// TwinCAT 3 PLC project Calvin
// ProgramVersion: 3.1.4023.0
// libraries:
//   Tc2_ModbusRTU, * (Beckhoff Automation GmbH)
//   Tc2_SerialCom, * (Beckhoff Automation GmbH)
//   Tc2_Standard, * (Beckhoff Automation GmbH)
//   Tc2_System, * (Beckhoff Automation GmbH)
//   Tc2_Utilities, * (Beckhoff Automation GmbH)
//   Tc3_Interfaces, * (Beckhoff Automation GmbH)
//   Tc3_Module, * (Beckhoff Automation GmbH)
//   Tc2_OpcUa,3.3.2.0,Beckhoff Automation GmbH
// project tree:
//   Data types/ E_OffOn.TcDUT, E_Alarms.TcDUT, E_MachineState.TcDUT, E_MBState.TcDUT, E_Status.TcDUT
//   GVLs/ Global_Constants.TcGVL, Global_Alarms.TcGVL, Global_Points.TcGVL, Global_Variables.TcGVL, Global_Variables_Tags.TcGVL
//   / PlcTask.TcTTO
//   POUs/Functions/ F_AnalogIn.TcPOU, F_Current.TcPOU, F_Voltage.TcPOU, F_Temperature.TcPOU
//   POUs/Function_Blocks/ FB_Temp_Control.TcPOU
//   POUs/ MAIN.TcPOU, P_AlarmCheck.TcPOU, P_HeaterControl.TcPOU, P_State_Machine.TcPOU, P_VFD_Test.TcPOU
// real-time tasks:
//   TASK PlcTask: cycle T#10ms, priority 20, ADS port 350
// I/O:
//   DEVICE Device 1 (EtherCAT), AmsNetId 10.12.1.55.2.1
//     Term 1 (EK1200) [EK1200-5000 EtherCAT Power supply (2A E-Bus)]
//       Term 2 (EL3318) [EL3318 8Ch. Ana Input Thermocouple (TC)]
//       Term 3 (EL3318) [EL3318 8Ch. Ana Input Thermocouple (TC)]
//       Term 4 (EL3318) [EL3318 8Ch. Ana Input Thermocouple (TC)]
//       Term 5 (EL3314) [EL3314 4Ch. Ana. Input Thermocouple (TC)]
//       Term 6 (EL3058) [EL3058 8Ch. Ana. Input 4-20mA]
//       Term 7 (EL3058) [EL3058 8Ch. Ana. Input 4-20mA]
//       Term 8 (EL3058) [EL3058 8Ch. Ana. Input 4-20mA]
//       Term 9 (EL3058) [EL3058 8Ch. Ana. Input 4-20mA]
//       Term 10 (EL3058) [EL3058 8Ch. Ana. Input 4-20mA]
//       Term 11 (EL9410) [EL9410 E-Bus Power Supplier  (Diagnostics)]
//       Term 12 (EL4122) [EL4122 2Ch. Ana. Output  4-20mA, 16bit]
//       Term 13 (EL4122) [EL4122 2Ch. Ana. Output  4-20mA, 16bit]
//       Term 14 (EL4122) [EL4122 2Ch. Ana. Output  4-20mA, 16bit]
//       Term 15 (EL4122) [EL4122 2Ch. Ana. Output  4-20mA, 16bit]
//       Term 16 (EL4122) [EL4122 2Ch. Ana. Output  4-20mA, 16bit]
//       Term 17 (EL1889) [EL1889 16Ch. Dig. Input 24V, 3ms, negative]
//       Term 18 (EL1889) [EL1889 16Ch. Dig. Input 24V, 3ms, negative]
//       Term 19 (EL9410) [EL9410 E-Bus Power Supplier  (Diagnostics)]
//       Term 20 (EL2088) [EL2088 8Ch. Dig. Output 24V, 0.5A, switching to negative]
//       Term 21 (EL2088) [EL2088 8Ch. Dig. Output 24V, 0.5A, switching to negative]
//       Term 22 (EL2088) [EL2088 8Ch. Dig. Output 24V, 0.5A, switching to negative]
//       Term 23 (EL2088) [EL2088 8Ch. Dig. Output 24V, 0.5A, switching to negative]
//       Term 24 (EL2008) [EL2008 8Ch. Dig. Output 24V, 0.5A]
//       Term 25 (EL6021) [EL6021 Interface (RS422/485)]
//       Term 26 (EL6021) [EL6021 Interface (RS422/485)]
//       Term 27 (EL2008) [EL2008 8Ch. Dig. Output 24V, 0.5A]
//       Term 28 (EL9011) [EL9011 End Terminal]
//   DEVICE Device 2 (NOV-DP-RAM)
//     Box 29 (Retain Handler)
// variable links:
//   Calvin/Calvin Instance <-> Device 1 (EtherCAT)/Term 1 (EK1200)/Term 10 (EL3058)
//     PlcTask Inputs/Global_Variables.IT_3 <-> AI Standard Channel 1/Value
//     PlcTask Inputs/Global_Variables.VT_1 <-> AI Standard Channel 2/Value
//     PlcTask Inputs/Global_Variables.VT_2 <-> AI Standard Channel 3/Value
//     PlcTask Inputs/Global_Variables.VT_3 <-> AI Standard Channel 4/Value
//     PlcTask Inputs/Global_Variables.ZT_1302B <-> AI Standard Channel 5/Value
//   Calvin/Calvin Instance <-> Device 1 (EtherCAT)/Term 1 (EK1200)/Term 12 (EL4122)
//     PlcTask Outputs/Global_Variables.IP_1102A <-> Channel 1/Output
//     PlcTask Outputs/Global_Variables.IP_1102B <-> Channel 2/Output
//   Calvin/Calvin Instance <-> Device 1 (EtherCAT)/Term 1 (EK1200)/Term 13 (EL4122)
//     PlcTask Outputs/Global_Variables.HS_1102_Out <-> Channel 2/Output
//     PlcTask Outputs/Global_Variables.IP_1101 <-> Channel 1/Output
//   Calvin/Calvin Instance <-> Device 1 (EtherCAT)/Term 1 (EK1200)/Term 14 (EL4122)
//     PlcTask Outputs/Global_Variables.HT_2_CTRL <-> Channel 1/Output
//     PlcTask Outputs/Global_Variables.HT_3_CTRL <-> Channel 2/Output
//   Calvin/Calvin Instance <-> Device 1 (EtherCAT)/Term 1 (EK1200)/Term 15 (EL4122)
//     PlcTask Outputs/Global_Variables.HT_4_CTRL <-> Channel 1/Output
//     PlcTask Outputs/Global_Variables.HT_5_CTRL <-> Channel 2/Output
//   Calvin/Calvin Instance <-> Device 1 (EtherCAT)/Term 1 (EK1200)/Term 16 (EL4122)
//     PlcTask Outputs/Global_Variables.HT_6_CTRL <-> Channel 1/Output
//     PlcTask Outputs/Global_Variables.IP_1302B <-> Channel 2/Output
//   Calvin/Calvin Instance <-> Device 1 (EtherCAT)/Term 1 (EK1200)/Term 17 (EL1889)
//     PlcTask Inputs/Global_Variables.ZSH_1101A <-> Channel 4/Input
//     PlcTask Inputs/Global_Variables.ZSH_1103A <-> Channel 8/Input
//     PlcTask Inputs/Global_Variables.ZSH_1301A <-> Channel 14/Input
//     PlcTask Inputs/Global_Variables.ZSH_1302A <-> Channel 16/Input
//     PlcTask Inputs/Global_Variables.ZSH_1101B <-> Channel 6/Input
//     PlcTask Inputs/Global_Variables.ZSH_1103B <-> Channel 10/Input
//     PlcTask Inputs/Global_Variables.ZSH_1107 <-> Channel 2/Input
//     PlcTask Inputs/Global_Variables.ZSH_1300 <-> Channel 12/Input
//     PlcTask Inputs/Global_Variables.ZSL_1101A <-> Channel 3/Input
//     PlcTask Inputs/Global_Variables.ZSL_1103A <-> Channel 7/Input
//     PlcTask Inputs/Global_Variables.ZSL_1301A <-> Channel 13/Input
//     PlcTask Inputs/Global_Variables.ZSL_1302A <-> Channel 15/Input
//     PlcTask Inputs/Global_Variables.ZSL_1101B <-> Channel 5/Input
//     PlcTask Inputs/Global_Variables.ZSL_1103B <-> Channel 9/Input
//     PlcTask Inputs/Global_Variables.ZSL_1107 <-> Channel 1/Input
//     PlcTask Inputs/Global_Variables.ZSL_1300 <-> Channel 11/Input
//   Calvin/Calvin Instance <-> Device 1 (EtherCAT)/Term 1 (EK1200)/Term 18 (EL1889)
//     PlcTask Inputs/Global_Variables.LSH_1201 <-> Channel 6/Input
//     PlcTask Inputs/Global_Variables.LSH_1202 <-> Channel 8/Input
//     PlcTask Inputs/Global_Variables.LSH_1300A <-> Channel 12/Input
//     PlcTask Inputs/Global_Variables.LSL_1201 <-> Channel 5/Input
//     PlcTask Inputs/Global_Variables.LSL_1202 <-> Channel 7/Input
//     PlcTask Inputs/Global_Variables.LSL_1300A <-> Channel 11/Input
//     PlcTask Inputs/Global_Variables.ZSH_1104 <-> Channel 10/Input
//     PlcTask Inputs/Global_Variables.ZSH_1301B <-> Channel 4/Input
//     PlcTask Inputs/Global_Variables.ZSL_1104 <-> Channel 9/Input
//     PlcTask Inputs/Global_Variables.ZSL_1301B <-> Channel 3/Input
//   Calvin/Calvin Instance <-> Device 1 (EtherCAT)/Term 1 (EK1200)/Term 2 (EL3318)
//     PlcTask Inputs/Global_Variables.TI_1001 <-> TC Channel 6/Value
//     PlcTask Inputs/Global_Variables.TI_1101 <-> TC Channel 7/Value
//     PlcTask Inputs/Global_Variables.TI_1301 <-> TC Channel 8/Value
//     PlcTask Inputs/Global_Variables.TI_1001_Error <-> TC Channel 6/Status/Error
//     PlcTask Inputs/Global_Variables.TI_1101_Error <-> TC Channel 7/Status/Error
//     PlcTask Inputs/Global_Variables.TI_1301_Error <-> TC Channel 8/Status/Error
//     PlcTask Inputs/Global_Variables.TI_1100A <-> TC Channel 2/Value
//     PlcTask Inputs/Global_Variables.TI_1102A <-> TC Channel 1/Value
//     PlcTask Inputs/Global_Variables.TI_1100A_Error <-> TC Channel 2/Status/Error
//     PlcTask Inputs/Global_Variables.TI_1102A_Error <-> TC Channel 1/Status/Error
//     PlcTask Inputs/Global_Variables.TI_1100B <-> TC Channel 3/Value
//     PlcTask Inputs/Global_Variables.TI_1102B <-> TC Channel 5/Value
//     PlcTask Inputs/Global_Variables.TI_1100B_Error <-> TC Channel 3/Status/Error
//     PlcTask Inputs/Global_Variables.TI_1102B_Error <-> TC Channel 5/Status/Error
//     PlcTask Inputs/Global_Variables.TI_1100C <-> TC Channel 4/Value
//     PlcTask Inputs/Global_Variables.TI_1100C_Error <-> TC Channel 4/Status/Error
//   Calvin/Calvin Instance <-> Device 1 (EtherCAT)/Term 1 (EK1200)/Term 20 (EL2088)
//     PlcTask Outputs/Global_Variables.HS_1200 <-> Channel 3/Output
//     PlcTask Outputs/Global_Variables.HS_1201 <-> Channel 4/Output
//     PlcTask Outputs/Global_Variables.HS_1202 <-> Channel 7/Output
//     PlcTask Outputs/Global_Variables.HS_1301 <-> Channel 2/Output
//     PlcTask Outputs/Global_Variables.HS_1300A <-> Channel 8/Output
//     PlcTask Outputs/Global_Variables.HT_1_RELAY <-> Channel 5/Output
//     PlcTask Outputs/Global_Variables.HT_2_RELAY <-> Channel 6/Output
//     PlcTask Outputs/Global_Variables.YL_1001 <-> Channel 1/Output
//   Calvin/Calvin Instance <-> Device 1 (EtherCAT)/Term 1 (EK1200)/Term 21 (EL2088)
//     PlcTask Outputs/Global_Variables.HS_1101A <-> Channel 8/Output
//     PlcTask Outputs/Global_Variables.HS_1107 <-> Channel 7/Output
//     PlcTask Outputs/Global_Variables.HS_1203 <-> Channel 3/Output
//     PlcTask Outputs/Global_Variables.HS_1305 <-> Channel 4/Output
//     PlcTask Outputs/Global_Variables.HT_3_RELAY <-> Channel 1/Output
//     PlcTask Outputs/Global_Variables.HT_4_RELAY <-> Channel 2/Output
//     PlcTask Outputs/Global_Variables.HT_5_RELAY <-> Channel 5/Output
//     PlcTask Outputs/Global_Variables.HT_6_RELAY <-> Channel 6/Output
//   Calvin/Calvin Instance <-> Device 1 (EtherCAT)/Term 1 (EK1200)/Term 22 (EL2088)
//     PlcTask Outputs/Global_Variables.HS_1101B <-> Channel 1/Output
//     PlcTask Outputs/Global_Variables.HS_1103B <-> Channel 3/Output
//     PlcTask Outputs/Global_Variables.HS_1300B <-> Channel 4/Output
//     PlcTask Outputs/Global_Variables.HS_1301B <-> Channel 8/Output
//     PlcTask Outputs/Global_Variables.HS_1102_Enable <-> Channel 7/Output
//     PlcTask Outputs/Global_Variables.HS_1103A <-> Channel 2/Output
//     PlcTask Outputs/Global_Variables.HS_1301A <-> Channel 5/Output
//     PlcTask Outputs/Global_Variables.HS_1302A <-> Channel 6/Output
//   Calvin/Calvin Instance <-> Device 1 (EtherCAT)/Term 1 (EK1200)/Term 23 (EL2088)
//     PlcTask Outputs/Global_Variables.AI_1102A_Pump <-> Channel 1/Output
//     PlcTask Outputs/Global_Variables.AI_1102A_Solenoid <-> Channel 2/Output
//     PlcTask Outputs/Global_Variables.AI_1102B_Pump <-> Channel 3/Output
//     PlcTask Outputs/Global_Variables.AI_1102B_Solenoid <-> Channel 4/Output
//     PlcTask Outputs/Global_Variables.HS_1104 <-> Channel 5/Output
//     PlcTask Outputs/Global_Variables.SV_1201 <-> Channel 8/Output
//     PlcTask Outputs/Global_Variables.YL_1002 <-> Channel 6/Output
//   Calvin/Calvin Instance <-> Device 1 (EtherCAT)/Term 1 (EK1200)/Term 24 (EL2008)
//     PlcTask Outputs/Global_Variables.LED1_Buzzer <-> Channel 3/Output
//     PlcTask Outputs/Global_Variables.LED2_Buzzer <-> Channel 6/Output
//     PlcTask Outputs/Global_Variables.LED1_G <-> Channel 2/Output
//     PlcTask Outputs/Global_Variables.LED2_G <-> Channel 5/Output
//     PlcTask Outputs/Global_Variables.LED1_R <-> Channel 1/Output
//     PlcTask Outputs/Global_Variables.LED2_R <-> Channel 4/Output
//     PlcTask Outputs/Global_Variables.LED3_R <-> Channel 7/Output
//     PlcTask Outputs/Global_Variables.LED3_Y <-> Channel 8/Output
//   Calvin/Calvin Instance <-> Device 1 (EtherCAT)/Term 1 (EK1200)/Term 25 (EL6021)
//     PlcTask Inputs/P_State_Machine.MBV_Master.InData/D[{0..21}] <-> COM Inputs/Data In {0..21}  (22 links)
//     PlcTask Inputs/P_State_Machine.MBV_Master.InData/Status <-> COM Inputs/Status
//     PlcTask Outputs/P_State_Machine.MBV_Master.OutData/Ctrl <-> COM Outputs/Ctrl
//     PlcTask Outputs/P_State_Machine.MBV_Master.OutData/D[{0..21}] <-> COM Outputs/Data Out {0..21}  (22 links)
//   Calvin/Calvin Instance <-> Device 1 (EtherCAT)/Term 1 (EK1200)/Term 27 (EL2008)
//     PlcTask Outputs/Global_Variables.LED3_Buzzer <-> Channel 2/Output
//     PlcTask Outputs/Global_Variables.LED3_G <-> Channel 1/Output
//   Calvin/Calvin Instance <-> Device 1 (EtherCAT)/Term 1 (EK1200)/Term 3 (EL3318)
//     PlcTask Inputs/Global_Variables.TI_1 <-> TC Channel 4/Value
//     PlcTask Inputs/Global_Variables.TI_1302 <-> TC Channel 1/Value
//     PlcTask Inputs/Global_Variables.TI_1303 <-> TC Channel 2/Value
//     PlcTask Inputs/Global_Variables.TI_1304 <-> TC Channel 3/Value
//     PlcTask Inputs/Global_Variables.TI_2 <-> TC Channel 5/Value
//     PlcTask Inputs/Global_Variables.TI_3 <-> TC Channel 6/Value
//     PlcTask Inputs/Global_Variables.TI_4 <-> TC Channel 7/Value
//     PlcTask Inputs/Global_Variables.TI_5 <-> TC Channel 8/Value
//     PlcTask Inputs/Global_Variables.TI_1302_Error <-> TC Channel 1/Status/Error
//     PlcTask Inputs/Global_Variables.TI_1303_Error <-> TC Channel 2/Status/Error
//     PlcTask Inputs/Global_Variables.TI_1304_Error <-> TC Channel 3/Status/Error
//     PlcTask Inputs/Global_Variables.TI_1_Error <-> TC Channel 4/Status/Error
//     PlcTask Inputs/Global_Variables.TI_2_Error <-> TC Channel 5/Status/Error
//     PlcTask Inputs/Global_Variables.TI_3_Error <-> TC Channel 6/Status/Error
//     PlcTask Inputs/Global_Variables.TI_4_Error <-> TC Channel 7/Status/Error
//     PlcTask Inputs/Global_Variables.TI_5_Error <-> TC Channel 8/Status/Error
//   Calvin/Calvin Instance <-> Device 1 (EtherCAT)/Term 1 (EK1200)/Term 4 (EL3318)
//     PlcTask Inputs/Global_Variables.TI_{6..12} <-> TC Channel {1..7}/Value  (7 links)
//     PlcTask Inputs/Global_Variables.TI_{6..12}_Error <-> TC Channel {1..7}/Status/Error  (7 links)
//   Calvin/Calvin Instance <-> Device 1 (EtherCAT)/Term 1 (EK1200)/Term 5 (EL3314)
//     PlcTask Inputs/Global_Variables.TI_{1103..1106} <-> TC Inputs Channel {1..4}/Value  (4 links)
//     PlcTask Inputs/Global_Variables.TI_{1103..1106}_Error <-> TC Inputs Channel {1..4}/Status/Error  (4 links)
//   Calvin/Calvin Instance <-> Device 1 (EtherCAT)/Term 1 (EK1200)/Term 6 (EL3058)
//     PlcTask Inputs/Global_Variables.DPT_1100 <-> AI Standard Channel 1/Value
//     PlcTask Inputs/Global_Variables.DPT_1102A <-> AI Standard Channel 4/Value
//     PlcTask Inputs/Global_Variables.DPT_1102B <-> AI Standard Channel 5/Value
//     PlcTask Inputs/Global_Variables.PI_1001 <-> AI Standard Channel 6/Value
//     PlcTask Inputs/Global_Variables.PI_1100 <-> AI Standard Channel 2/Value
//     PlcTask Inputs/Global_Variables.PI_1101 <-> AI Standard Channel 3/Value
//     PlcTask Inputs/Global_Variables.PI_1200 <-> AI Standard Channel 7/Value
//     PlcTask Inputs/Global_Variables.PI_1300 <-> AI Standard Channel 8/Value
//   Calvin/Calvin Instance <-> Device 1 (EtherCAT)/Term 1 (EK1200)/Term 7 (EL3058)
//     PlcTask Inputs/Global_Variables.FIC_1102 <-> AI Standard Channel 1/Value
//     PlcTask Inputs/Global_Variables.FI_1001 <-> AI Standard Channel 2/Value
//     PlcTask Inputs/Global_Variables.FI_1300 <-> AI Standard Channel 5/Value
//     PlcTask Inputs/Global_Variables.FI_1301 <-> AI Standard Channel 4/Value
//     PlcTask Inputs/Global_Variables.FI_1200_1 <-> AI Standard Channel 3/Value
//     PlcTask Inputs/Global_Variables.ZT_1101 <-> AI Standard Channel 8/Value
//     PlcTask Inputs/Global_Variables.ZT_1102A <-> AI Standard Channel 6/Value
//     PlcTask Inputs/Global_Variables.ZT_1102B <-> AI Standard Channel 7/Value
//   Calvin/Calvin Instance <-> Device 1 (EtherCAT)/Term 1 (EK1200)/Term 8 (EL3058)
//     PlcTask Inputs/Global_Variables.AI_1102A <-> AI Standard Channel 3/Value
//     PlcTask Inputs/Global_Variables.AI_1102B <-> AI Standard Channel 4/Value
//     PlcTask Inputs/Global_Variables.AI_1301 <-> AI Standard Channel 5/Value
//     PlcTask Inputs/Global_Variables.LIC_1300 <-> AI Standard Channel 2/Value
//     PlcTask Inputs/Global_Variables.LI_1204 <-> AI Standard Channel 1/Value
//     PlcTask Inputs/Global_Variables.MI_1102A <-> AI Standard Channel 8/Value
//   Calvin/Calvin Instance <-> Device 1 (EtherCAT)/Term 1 (EK1200)/Term 9 (EL3058)
//     PlcTask Inputs/Global_Variables.FI_1200_2 <-> AI Standard Channel 1/Value
//     PlcTask Inputs/Global_Variables.FI_1200_3 <-> AI Standard Channel 2/Value
//     PlcTask Inputs/Global_Variables.FI_1201_1 <-> AI Standard Channel 4/Value
//     PlcTask Inputs/Global_Variables.FI_1201_2 <-> AI Standard Channel 5/Value
//     PlcTask Inputs/Global_Variables.FI_1201_3 <-> AI Standard Channel 6/Value
//     PlcTask Inputs/Global_Variables.IT_1 <-> AI Standard Channel 7/Value
//     PlcTask Inputs/Global_Variables.IT_2 <-> AI Standard Channel 8/Value
//     PlcTask Inputs/Global_Variables.MI_1102B <-> AI Standard Channel 3/Value
//   Calvin/Calvin Instance <-> Device 2 (NOV-DP-RAM)/Box 29 (Retain Handler)
//     PlcTask Retains/P_State_Machine.gpdiCycle_Count <-> Retains/P_State_Machine.gpdiCycle_Count_[851]

CONFIGURATION Calvin
    RESOURCE PLC ON TwinCAT3
        TASK PlcTask(INTERVAL := T#10ms, PRIORITY := 20);
        PROGRAM MAIN WITH PlcTask : MAIN;
    END_RESOURCE
END_CONFIGURATION

// ---- Data types/E_OffOn.TcDUT
// Calvin - E_OffOn
// Rev 1.00 - March 23, 2023

TYPE E_OffOn :
(
	eOFF 	:= 1,
	eON		:= 2
);
END_TYPE

// ---- Data types/E_Alarms.TcDUT
// Calvin - E_Alarms
// Rev 1.00 - May 25, 2023

TYPE E_Alarms :
(
	eNo_Alarms							:= 0,
	eWarmup_Alarm,					
	eEvacuation_Alarm,					
	eSteamBypass_Alarm,					
	eDesorption_Alarm,					
	eRepressurization_Alarm,					
	eAdsorption_Alarm,					
	eSystem_Alarm,					
	eTC_Alarm,					
	eT09_Alarm,					
	eT10_Alarm,					
	eT11_Alarm,					
	eT12_Alarm,					
	eT13_Alarm,					
	eT14_Alarm,					
	eT15_Alarm,					
	eT16_Alarm,					
	eT17_Alarm,					
	eT18_Alarm,					
	eT19_Alarm,					
	eT20_Alarm,					
	eTimeout_Alarm,							// 21		
	e22_Error,		
	eReactorBackflow_Error,			
	eEvacTargetPressure_Error,		
	eCondensateLS_Error,			
	eDesorpNominalPressure_Error,	
	eDesorpCO2Conc_Error,			
	eReactorCooling_Error,			
	eReactorHighPressure_Error,		
	eReactorLowPressure_Error,		
	eReactorHighTemp_Error,			
	eReactorLowTemp_Error,			
	eHighLevel_Error,				
	eLowLevel_Error,				
	eVacuumHighTemp_Error,			
	eCondenserNoFlow_Error,			
	eHeatTrace_Error,				
	eSteamLS_Error,					
	eHeatTraceTimeout_Error,		
	eDPT_311_Error,					
	eDPTError						
);                                  
END_TYPE

// ---- Data types/E_MachineState.TcDUT
// Calvin - E_MachineState
// Rev 1.00 - April 26, 2023

TYPE E_MachineState :
(
	eIdle						:= 0,
	eWarmup,
	eEvacuation,
	eSteamBypass,
	eDesorption,
	eRepressurization,
	eAdsorption,
	eReset,
	ePause,
	eSystemError
);
END_TYPE

// ---- Data types/E_MBState.TcDUT
// Calvin - E_MBState
// Rev 1.00 - April 6, 2023

TYPE E_MBState :
(
	eMBIdle			 			:= 0,
	eMBReadCoils,
	eMBReadInputStatus,
	eMBReadRegs,
	eMBReadInputRegs,
	eMBWriteSingleCoil,
	eMBWriteSingleReg,
	eMBWriteMultipleCoils,
	eMBWriteRegs
);
END_TYPE

// ---- Data types/E_Status.TcDUT
// Calvin - E_Status
// Rev 1.00 - April 27, 2023

TYPE E_Status :
(
	eStart_Warm_Up						:= 0,
	eWarmup_Running,							// 1
	eStart_Reactor_Reset,						// 2
	eSystem_Ready,								// 3
	eEvacuation_Running,						// 4
	eSteamBypass_Running,						// 5
	eRepressurization_Running,					// 6
	eDesorption_Running,						// 7
	eAdsorption_Running,						// 8
	e9,
	eStopping_Process,							// 10
	eStopping_Warmup,							// 11
	eStopping_Evacuation,						// 12
	eStopping_SteamBypass,						// 13
	eStopping_Repressurization,					// 14
	eStopping_Desorption,						// 15
	eStopping_Adsorption,						// 16
	e17,
	eCycle_Error,								// 18
	e19,
	e20,
	eTest_Running,								// 21
	eEvacuation_Process_Error,					// 22
	eSteamBypass_Process_Error,					// 23
	eRepressurization_Process_Error,			// 24
	eDesorption_Process_Error,					// 25
	eAdsorption_Process_Error,					// 26
	e27,
	e28,
	e29,
	eEvacuation_Complete,						// 30
	eSteamBypass_Complete,						// 31
	eRepressurization_Complete,					// 32
	eDesorption_Complete,						// 33
	eAdsorption_Complete						// 34
);
END_TYPE

// ---- GVLs/Global_Constants.TcGVL
// Calvin - Global_Constants
// Rev 1.00 - September 22, 2023

VAR_GLOBAL
	PID_CYCLE_TIME									: REAL 		:= 0.01;		// PID cycle time for heaters
	OUTPUT_MIN										: REAL		:= 200;			// Minimum output needed to energize solid state heater relay
	PERCENT_FACTOR									: REAL		:= 327.67;		// Factor to convert input to output percentage
	ALARM_COUNT										: INT		:= 100;			// Number of possible alarms
	PRESSURE_CUTOFF									: REAL		:= 0.8;
	DEFAULT_STEP_TIME								: REAL		:= 20000;		// 20 seconds default time
	SECONDS											: REAL		:= 1000;
	MINUTES											: REAL		:= 60000;
	RESET_TIME										: REAL		:= 2000;
	
	CONDENSER_LEVEL_REFILL							: REAL		:= 20;											// 09/21/23 PS
	CONDENSER_LEVEL_LOW_LIMIT						: REAL		:= 12;											// 09/21/23 PS
	CONDENSER_LEVEL_HIGH_LIMIT						: REAL		:= 60;											// 09/21/23 PS
	VACUUM_TANK_DRAIN_TIME							: REAL		:= 60;											// 09/22/23 PS
	
	MB_VFD_ENABLE_ADDR								: WORD		:= 8192;
	MB_VFD_FREQ_ADDR								: WORD		:= 8193;
	MB_VFD_BLOCK_ADDR								: WORD		:= 2315;
	MODBUS_TIMEOUT									: TIME 		:= T#1S;
	 
	BV_OPEN_MAX										: REAL		:= 100.0;                               	
	BV_OPEN_POS_THRESHOLD							: REAL		:= 10.0;			// Percent that valve must be within open position to trigger open status
	BV_CLOSED_POS_THRESHOLD							: REAL		:= 2;				// Percent that valve must be within closed position to trigger closed status
	                                					
END_VAR

// ---- GVLs/Global_Alarms.TcGVL
// Calvin - Global_Alarms
// Rev 1.00 - September 22, 2023

VAR_GLOBAL
	gbAlarmsLoaded									: BOOL;
	gbRunVFD										: BOOL;
	giActiveAlarm									: INT;
	gbAlarms										: ARRAY[0..100] OF BOOL;
	gsAlarms										: ARRAY[0..100] OF STRING;
	gsAlarmInfo										: ARRAY[0..100] OF STRING;
	gsTempAlarm										: STRING;

	gsTI_1101Error									: STRING	:= '-TI_1101 sensor error';						// 09/20/23 PS
	gsLowCondenserLevel								: STRING	:= '-Condenser level low';						// 09/07/23 PS
	gsTK1300HighLevel								: STRING	:= '-TK_1300 level high';
	
	gsBoilerPressureLow								: STRING	:= '-Boiler pressure low';
	gsDrainNotClear									: STRING	:= '-Drain not clear';
	gsValvesNotClosed								: STRING	:= '-Valves not closed';
	gsValvesNotOpen									: STRING	:= '-Valves not open';
	gsLRPCoolingFlowLow								: STRING	:= '-LRP cooling flow low';
	gsTargetPressureHigh							: STRING	:= '-Target pressure high';
	gsPI_1300OutOfRange								: STRING	:= '-PI_1300 out of range';
	gsPI_1100OutOfRange								: STRING	:= '-PI_1100 out of range';
	gsPI_1100PressureLow							: STRING	:= '-PI_1100 pressure low';
	gsPI_1101PressureLow							: STRING	:= '-PI_1101 pressure low';
	gsPI_1001PressureLow							: STRING	:= '-PI_1001 pressure low';
	gsVacuumLeak									: STRING	:= '-Vacuum leak';
	gsSteamFlowLow									: STRING	:= '-Steam flow low';
	gsSteamTempLow									: STRING	:= '-Steam temperature low';
	gsSteamTempError								: STRING	:= '-Steam temperature sensor error';
	gsLimitSwitchError								: STRING	:= '-Limit swtich error';
	gsValveOutOfRange								: STRING	:= '-Valve out of range';
	gsReactorPressureLow							: STRING	:= '-Reactor pressure low';
	gsThermocoupleError								: STRING	:= '-Thermocouple error';
	gsSorbentOverTemp								: STRING	:= '-Sorbent over temperature';
	gsTempOutOfRange								: STRING	:= '-Temperature out of range';
	gsNoAirFlow										: STRING	:= '-No air flow';
	gsCO2DifferentialError							: STRING	:= '-CO2 differential error';
	gsFanStillRunning								: STRING	:= '-Fan still runiing';
	gsFileSaveError									: STRING	:= 'File save error';
	
	ALARM_00										: STRING	:= '00/No Alarms';								// These must correspond to E_Alarms values
	ALARM_01										: STRING	:= '01/ Warmup Error - ';
	ALARM_02										: STRING	:= '02/ Evacuation Error - ';
	ALARM_03										: STRING	:= '03/ Steam Bypass Error - ';
	ALARM_04										: STRING	:= '04/ Desorption Error - ';
	ALARM_05										: STRING	:= '05/ Repressurization Error - ';
	ALARM_06										: STRING	:= '06/ Adsorption Error - ';
	ALARM_07										: STRING	:= '07/ System Error - ';
	ALARM_08										: STRING	:= '08/ Thermocouple Error';
	ALARM_09										: STRING	:= '09/Alarm';
	ALARM_10										: STRING	:= '10/Alarm';
	ALARM_11										: STRING	:= '11/Alarm';
	ALARM_12										: STRING	:= '12/Alarm';
	ALARM_13										: STRING	:= '13/Alarm';
	ALARM_14										: STRING	:= '14/Alarm';
	ALARM_15										: STRING	:= '15/Alarm';
	ALARM_16										: STRING	:= '16/Alarm';
	ALARM_17										: STRING	:= '17/Alarm';
	ALARM_18										: STRING	:= '18/Alarm';
	ALARM_19										: STRING	:= '19/Alarm';
	ALARM_20										: STRING	:= '20/Alarm';
	ALARM_21										: STRING	:= '21Timeout Error';
	ALARM_22										: STRING	:= '22Alarm';
	ALARM_23										: STRING	:= '23Alarm';
	ALARM_24										: STRING	:= '24Alarm';
	ALARM_25										: STRING	:= '25Alarm';
	ALARM_26										: STRING	:= '26Alarm';
	ALARM_27										: STRING	:= '27Alarm';
	ALARM_28										: STRING	:= '28Alarm';
	ALARM_29										: STRING	:= '29Alarm';
	ALARM_30										: STRING	:= '30Alarm';
	ALARM_31										: STRING	:= '31Alarm';
	ALARM_32										: STRING	:= '32Alarm';
	ALARM_33										: STRING	:= '33Alarm';
	ALARM_34										: STRING	:= '34Alarm';
	ALARM_35										: STRING	:= '35Alarm';
	ALARM_36										: STRING	:= '36Alarm';
	ALARM_37										: STRING	:= '37Alarm';
	ALARM_38										: STRING	:= '38Alarm';
	ALARM_39										: STRING	:= '39Alarm';
	ALARM_40										: STRING	:= '40Alarm';
	ALARM_41										: STRING	:= '41Alarm';
	ALARM_42										: STRING	:= '42Alarm';
	ALARM_43										: STRING	:= '43Alarm';
	ALARM_44										: STRING	:= '44Alarm';
	ALARM_45										: STRING	:= '45Alarm';
	ALARM_46										: STRING	:= '46Alarm';
	ALARM_47										: STRING	:= '47Alarm';
	ALARM_48										: STRING	:= '48Alarm';
	ALARM_49										: STRING	:= '49Alarm';
	ALARM_50										: STRING	:= '50Alarm';
END_VAR

// ---- GVLs/Global_Points.TcGVL
// Calvin - Global_Points
// Rev 1.00 - May 11, 2023

VAR_GLOBAL
	// Analog Input Sensor Ranges      			
	DPT_1102A_LOW									: REAL		:= 0.0;
	DPT_1102A_HIGH									: REAL		:= 10.0;
	DPT_1102A_MIN									: REAL		:= 0.01;
	DPT_1102A_OFFSET								: REAL		:= 0.0;
	FIC_1102_LOW									: REAL		:= 0.0;
	FIC_1102_HIGH									: REAL		:= 1500.0;
	FIC_1102_MIN									: REAL		:= 10.0;
	FIC_1102_OFFSET									: REAL		:= 0.0;
	AI_1102A_LOW									: REAL		:= 0.0;
	AI_1102A_HIGH									: REAL		:= 100.0;
	AI_1102A_MIN									: REAL		:= 0.01;
	AI_1102A_OFFSET									: REAL		:= 0.0;
	MI_1102A_LOW									: REAL		:= 0.0;
	MI_1102A_HIGH									: REAL		:= 100.0;
	MI_1102A_MIN									: REAL		:= 0.01;
	MI_1102A_OFFSET									: REAL		:= 0.0;
	ZT_1102A_LOW									: REAL		:= 0.0;
	ZT_1102A_HIGH									: REAL		:= 100.0;
	ZT_1102A_MIN									: REAL		:= 0.01;
	ZT_1102A_OFFSET									: REAL		:= 0.0;
	PI_1100_LOW										: REAL		:= 0.0;
	PI_1100_HIGH									: REAL		:= 100.0;
	PI_1100_MIN										: REAL		:= 0.01;
	PI_1100_OFFSET									: REAL		:= 0.0;
	DPT_1100_LOW									: REAL		:= -3.0;
	DPT_1100_HIGH									: REAL		:= 3.0;
	DPT_1100_MIN									: REAL		:= 0.01;
	DPT_1100_OFFSET									: REAL		:= 0.0;
	ZT_1102B_LOW									: REAL		:= 0.0;
	ZT_1102B_HIGH									: REAL		:= 100.0;
	ZT_1102B_MIN									: REAL		:= 0.01;
	ZT_1102B_OFFSET									: REAL		:= 0.0;
	AI_1102B_LOW									: REAL		:= 0.0;
	AI_1102B_HIGH									: REAL		:= 100.0;
	AI_1102B_MIN									: REAL		:= 0.01;
	AI_1102B_OFFSET									: REAL		:= 0.0;
	MI_1102B_LOW									: REAL		:= 0.0;
	MI_1102B_HIGH									: REAL		:= 100.0;
	MI_1102B_MIN									: REAL		:= 0.01;
	MI_1102B_OFFSET									: REAL		:= 0.0;
	DPT_1102B_LOW									: REAL		:= 0.0;
	DPT_1102B_HIGH									: REAL		:= 5.0;
	DPT_1102B_MIN									: REAL		:= 0.01;
	DPT_1102B_OFFSET								: REAL		:= 0.0;
	FI_1200_1_LOW									: REAL		:= 0.0;
	FI_1200_1_HIGH									: REAL		:= 1500.0;
	FI_1200_1_MIN									: REAL		:= 10.0;
	FI_1200_1_OFFSET								: REAL		:= 0.0;
	FI_1200_2_LOW									: REAL		:= 0.0;
	FI_1200_2_HIGH									: REAL		:= 1500.0;
	FI_1200_2_MIN									: REAL		:= 10.0;
	FI_1200_2_OFFSET								: REAL		:= 0.0;
	FI_1200_3_LOW									: REAL		:= 0.0;
	FI_1200_3_HIGH									: REAL		:= 1500.0;
	FI_1200_3_MIN									: REAL		:= 10.0;
	FI_1200_3_OFFSET								: REAL		:= 0.0;
	FI_1201_1_LOW									: REAL		:= 0.0;
	FI_1201_1_HIGH									: REAL		:= 1500.0;
	FI_1201_1_MIN									: REAL		:= 10.0;
	FI_1201_1_OFFSET								: REAL		:= 0.0;
	FI_1201_2_LOW									: REAL		:= 0.0;
	FI_1201_2_HIGH									: REAL		:= 1500.0;
	FI_1201_2_MIN									: REAL		:= 10.0;
	FI_1201_2_OFFSET								: REAL		:= 0.0;
	FI_1201_3_LOW									: REAL		:= 0.0;
	FI_1201_3_HIGH									: REAL		:= 1500.0;
	FI_1201_3_MIN									: REAL		:= 10.0;
	FI_1201_3_OFFSET								: REAL		:= 0.0;
	PI_1200_LOW										: REAL		:= 0.0;
	PI_1200_HIGH									: REAL		:= 100.0;
	PI_1200_MIN										: REAL		:= 0.01;
	PI_1200_OFFSET									: REAL		:= 0.0;
	PI_1001_LOW										: REAL		:= 0.0;
	PI_1001_HIGH									: REAL		:= 100.0;
	PI_1001_MIN										: REAL		:= 0.01;
	PI_1001_OFFSET									: REAL		:= 0.0;
	FI_1001_LOW										: REAL		:= 0.0;
	FI_1001_HIGH									: REAL		:= 100.0;
	FI_1001_MIN										: REAL		:= 0.01;
	FI_1001_OFFSET									: REAL		:= 0.0;
	ZT_1101_LOW										: REAL		:= 0.0;
	ZT_1101_HIGH									: REAL		:= 100.0;
	ZT_1101_MIN										: REAL		:= 0.01;
	ZT_1101_OFFSET									: REAL		:= 0.0;
	PI_1101_LOW										: REAL		:= 0.0;
	PI_1101_HIGH									: REAL		:= 100.0;
	PI_1101_MIN		 								: REAL		:= 0.01;
	PI_1101_OFFSET									: REAL		:= 0.0;
	LI_1204_LOW										: REAL		:= 0.0;
	LI_1204_HIGH									: REAL		:= 100.0;
	LI_1204_MIN										: REAL		:= 0.01;
	LI_1204_OFFSET									: REAL		:= 0.0;
	AI_1300_1_LOW									: REAL		:= 0.0;
	AI_1300_1_HIGH									: REAL		:= 100.0;
	AI_1300_1_MIN									: REAL		:= 0.01;
	AI_1300_1_OFFSET								: REAL		:= 0.0;
	AI_1300_2_LOW									: REAL		:= 0.0;
	AI_1300_2_HIGH									: REAL		:= 100.0;
	AI_1300_2_MIN									: REAL		:= 0.01;
	AI_1300_2_OFFSET								: REAL		:= 0.0;
	AI_1300_3_LOW									: REAL		:= 0.0;
	AI_1300_3_HIGH									: REAL		:= 100.0;
	AI_1300_3_MIN									: REAL		:= 0.01;
	AI_1300_3_OFFSET								: REAL		:= 0.0;
	PI_1300_LOW										: REAL		:= 0.0;
	PI_1300_HIGH									: REAL		:= 100.0;
	PI_1300_MIN										: REAL		:= 0.01;
	PI_1300_OFFSET									: REAL		:= 0.0;
	LIC_1300_LOW									: REAL		:= 0.0;
	LIC_1300_HIGH									: REAL		:= 100.0;
	LIC_1300_MIN									: REAL		:= 0.01;
	LIC_1300_OFFSET									: REAL		:= 0.0;
	FI_1300_LOW										: REAL		:= 0.0;
	FI_1300_HIGH									: REAL		:= 100.0;
	FI_1300_MIN										: REAL		:= 0.01;
	FI_1300_OFFSET									: REAL		:= 0.0;
	FI_1301_LOW										: REAL		:= 0.0;
	FI_1301_HIGH									: REAL		:= 100.0;
	FI_1301_MIN										: REAL		:= 0.01;
	FI_1301_OFFSET									: REAL		:= 0.0;
	AI_1301_LOW										: REAL		:= 0.0;
	AI_1301_HIGH									: REAL		:= 100.0;
	AI_1301_MIN										: REAL		:= 0.01;
	AI_1301_OFFSET									: REAL		:= 0.0;
	ZT_1302B_LOW									: REAL		:= 0.0;
	ZT_1302B_HIGH									: REAL		:= 0.0;
	ZT_1302B_MIN									: REAL		:= 0.0;
	ZT_1302B_OFFSET									: REAL		:= 0.0;
	
	MI_2001_LOW										: REAL		:= 0.0;
	MI_2001_HIGH									: REAL		:= 100.0;
	MI_2001_MIN										: REAL		:= 0.01;
	MI_2001_OFFSET									: REAL		:= 0.0;
	TI_2001_LOW										: REAL		:= 0.0;
	TI_2001_HIGH									: REAL		:= 100.0;
	TI_2001_MIN										: REAL		:= 0.01;
	TI_2001_OFFSET									: REAL		:= 0.0;
	SI_2001_LOW										: REAL		:= 0.0;
	SI_2001_HIGH									: REAL		:= 100.0;
	SI_2001_MIN										: REAL		:= 0.01;
	SI_2001_OFFSET									: REAL		:= 0.0;
	ZI_2001_LOW										: REAL		:= 0.0;
	ZI_2001_HIGH									: REAL		:= 100.0;
	ZI_2001_MIN										: REAL		:= 0.01;
	ZI_2001_OFFSET									: REAL		:= 0.0;
	PI_2001_LOW										: REAL		:= 0.0;
	PI_2001_HIGH									: REAL		:= 100.0;
	PI_2001_MIN										: REAL		:= 0.01;
	PI_2001_OFFSET									: REAL		:= 0.0;

	ZXI_2002_LOW									: REAL		:= 0.0;
	ZXI_2002_HIGH									: REAL		:= 100.0;
	ZXI_2002_MIN									: REAL		:= 0.01;
	ZXI_2002_OFFSET									: REAL		:= 0.0;
	ZYI_2002_LOW									: REAL		:= 0.0;
	ZYI_2002_HIGH									: REAL		:= 100.0;
	ZYI_2002_MIN									: REAL		:= 0.01;
	ZYI_2002_OFFSET									: REAL		:= 0.0;
                        				
END_VAR

// ---- GVLs/Global_Variables.TcGVL
// Calvin - Global_Variables
// Rev 1.00 - September 20, 2023

VAR_GLOBAL
	eState											: E_MachineState;

	grHS_1102Out									: REAL;
	grSteamValveSP									: REAL;
	gbVFDTest										: BOOL;
	gbReadMBVFD										: BOOL;
	gbReadMBWeather									: BOOL;
	gbReadMBInclinometer							: BOOL;
	gbHS_1102ValvesOpen								: BOOL;
	gbHS_1102ValvesClosed							: BOOL;
	gbVacuumHolding									: BOOL;

	datain					AT %I*					: REAL;
	dataout					AT %Q*					: BYTE;

	// Reactor
	DPT_1102A				AT %I*					: INT;			// Reactor Filter Differential Pressure (-7.46 to 7.46 mbar)
	FIC_1102				AT %I*					: INT;			// Reactor Air flow
	AI_1102A				AT %I*					: INT;			// Reactor Inlet C02 (ppm)
	AI_1102A_Pump			AT %Q*					: BOOL;			// Inlet CO2 pump
	AI_1102A_Solenoid		AT %Q*					: BOOL;			// Inlet CO2 solenoid
	MI_1102A				AT %I*					: INT;			// Reactor Inlet H20 (ppm)
	ZT_1102A				AT %I*					: INT;			// Reactor Inlet Isolation Valve Input
	PI_1100					AT %I*					: INT;			// Reactor Pressure
	TI_1102A				AT %I*					: INT;			// Reactor Inlet Temperature
	TI_1102A_Error			AT %I*					: BOOL;			// Reactor Inlet Temperature Error
	bTI_1102A_ErrActive								: BOOL;
	TI_1100A				AT %I*					: INT;			// Reactor Sorbent Temperature A
	TI_1100A_Error			AT %I*					: BOOL;			// Reactor Sorbent Temperature A Error
	bTI_1100A_ErrActive								: BOOL;
	TI_1100B				AT %I*					: INT;			// Reactor Sorbent Temperature B
	TI_1100B_Error			AT %I*					: BOOL;			// Reactor Sorbent Temperature B Error
	bTI_1100B_ErrActive								: BOOL;
	TI_1100C				AT %I*					: INT;			// Reactor Sorbent Temperature C
	TI_1100C_Error			AT %I*					: BOOL;			// Reactor Sorbent Temperature C Error
	bTI_1100C_ErrActive								: BOOL;
	DPT_1100				AT %I*					: INT;			// Reactor Differential Pressure
	ZT_1102B				AT %I*					: INT;			// Reactor Outlet Isolation Valve Input
	TI_1102B				AT %I*					: INT;			// Reactor Outlet Temperature
	TI_1102B_Error			AT %I*					: BOOL;			// Reactor Outlet Temperature Error
	bTI_1102B_ErrActive								: BOOL;
	AI_1102B				AT %I*					: INT;			// Reactor Outlet C02 (ppm)
	AI_1102B_Pump			AT %Q*					: BOOL;			// Outlet CO2 pump
	AI_1102B_Solenoid		AT %Q*					: BOOL;			// Outlet CO2 solenoid
	MI_1102B				AT %I*					: INT;			// Reactor Outlet H20 (ppm)
	DPT_1102B				AT %I*					: INT;			// Reactor Fan Static Pressure
	IP_1102A				AT %Q*					: INT;			// Reactor Inlet Isolation Butterfly Valve Output
	IP_1102B				AT %Q*					: INT;			// Reactor Outlet Isolation Butterfly Valve Output
	HS_1104					AT %Q*					: BOOL;			// Reactor valve
	ZSH_1104				AT %I*					: BOOL;			// Reactor valve open
	ZSL_1104				AT %I*					: BOOL;			// Reactor valve closed
	TI_1103					AT %I*					: INT;			// Reactor Wall Temperature 1
	TI_1103_Error			AT %I*					: BOOL;			// Reactor Wall Temperature 1 Error
	bTI_1103_ErrActive								: BOOL;
	TI_1104					AT %I*					: INT;			// Reactor Wall Temperature 1
	TI_1104_Error			AT %I*					: BOOL;			// Reactor Wall Temperature 1 Error
	bTI_1104_ErrActive								: BOOL;
	TI_1105					AT %I*					: INT;			// Reactor Wall Temperature 1
	TI_1105_Error			AT %I*					: BOOL;			// Reactor Wall Temperature 1 Error
	bTI_1105_ErrActive								: BOOL;
	TI_1106					AT %I*					: INT;			// Reactor Wall Temperature 1
	TI_1106_Error			AT %I*					: BOOL;			// Reactor Wall Temperature 1 Error
	bTI_1106_ErrActive								: BOOL;
	
	// Steam
	FI_1200_1				AT %I*					: INT;			// Boiler Feed Flow
	FI_1200_2				AT %I*					: INT;			// Boiler Feed Flow
	FI_1200_3				AT %I*					: INT;			// Boiler Feed Flow
	FI_1201_1				AT %I*					: INT;			// Boiler Feed Flow
	FI_1201_2				AT %I*					: INT;			// Boiler Feed Flow
	FI_1201_3				AT %I*					: INT;			// Boiler Feed Flow
	PI_1200					AT %I*					: INT;			// Boiler Feed Water Pressure
	PI_1001					AT %I*					: INT;			// Boiler Steam Pressure
	TI_1001					AT %I*					: INT;			// Boiler Steam Temperature
	TI_1001_Error			AT %I*					: BOOL;			// Boiler Steam Temperature Error
	bTI_1001_ErrActive								: BOOL;
	FI_1001					AT %I*					: INT;			// Steam Line Pressure
	ZT_1101					AT %I*					: INT;			// Steam Control Valve Input
	PI_1101					AT %I*					: INT;			// Steam Line Pressure
	TI_1101					AT %I*					: INT;			// Steam Line Temperature
	TI_1101_Error			AT %I*					: BOOL;			// Steam Line Temperature Error
	bTI_1101_ErrActive								: BOOL;
	ZSH_1107				AT %I*					: BOOL;			// Steam Bypass Valve High Limit Switch
	ZSL_1107				AT %I*					: BOOL;			// Steam Bypass Valve Low Limit Switch
	ZSH_1101A				AT %I*					: BOOL;			// Reactor Steam Isolation Valve A High Limit Switch
	ZSL_1101A				AT %I*					: BOOL;			// Reactor Steam Isolation Valve A Low Limit Switch
	ZSH_1101B				AT %I*					: BOOL;			// Reactor Steam Isolation Valve B High Limit Switch
	ZSL_1101B				AT %I*					: BOOL;			// Reactor Steam Isolation Valve B Low Limit Switch
	IP_1101					AT %Q*					: INT;			// Steam Control Valve Output
	YL_1001					AT %Q*					: BOOL;			// Boiler Power Contactor
	YL_1002					AT %Q*					: BOOL;			// Boiler Power Contactor
	HS_1107					AT %Q*					: BOOL;			// Steam Bypass Valve Output
	HS_1101A				AT %Q*					: BOOL;			// Reactor Steam Isolation Valve A
	HS_1101B				AT %Q*					: BOOL;			// Reactor Steam Isolation Valve B
	                                            	
	// Condensate
	HS_1201					AT %Q*					: BOOL;			// Reactor Drain Pump
	LSH_1201				AT %I*					: BOOL;			// Reactor Drain Level High
	LSL_1201				AT %I*					: BOOL;			// Reactor Drain Level Low
	HS_1103A				AT %Q*					: BOOL;			// Reactor To Vacuum Isolation Valve A
	ZSH_1103A				AT %I*					: BOOL;			// Reactor To Vacuum Isolation Valve A High Limit Switch
	ZSL_1103A				AT %I*					: BOOL;			// Reactor To Vacuum Isolation Valve A Low Limit Switch
	HS_1103B				AT %Q*					: BOOL;			// Reactor To Vacuum Isolation Valve B
	ZSH_1103B				AT %I*					: BOOL;			// Reactor To Vacuum Isolation Valve B High Limit Switch
	ZSL_1103B				AT %I*					: BOOL;			// Reactor To Vacuum Isolation Valve B Low Limit Switch
	HS_1203					AT %Q*					: BOOL;			// Condenser Heater Motor
	HS_1202					AT %Q*					: BOOL;			// Separator Drain Pump
	LSH_1202				AT %I*					: BOOL;			// Separator Drain Level High Switch
	LSL_1202				AT %I*					: BOOL;			// Separator Drain Level Low Switch
	LI_1204					AT %I*					: INT;			// Condensate Tank Level
	HS_1200					AT %Q*					: BOOL;			// Condensate/Boiler Feed Pump
	SV_1201					AT %Q*					: BOOL;			// Refill valve													// 09/19/23 PS
	ZSH_1202				AT %I*					: BOOL;			// Refill valve													// 09/19/23 PS
	ZSL_1202				AT %I*					: BOOL;			// Refill valve													// 09/19/23 PS
                                                	
	// Vacuum
	HS_1302A				AT %Q*					: BOOL;			// Vacuum Desorb Valve
	ZSH_1302A				AT %I*					: BOOL;			// Vacuum Desorb Valve High Limit Switch
	ZSL_1302A				AT %I*					: BOOL;			// Vacuum Desorb Valve Low Limit Switch
	IP_1302B				AT %Q*					: INT;			// Ambient Steam Desorption Valve
	ZT_1302B				AT %I*					: INT;			// Ambient Steam Desorption Valve feedback
	PI_1300					AT %I*					: INT;			// Vacuum System Pressure
	HS_1301A				AT %Q*					: BOOL;			// Eductor Valve
	ZSH_1301A				AT %I*					: BOOL;			// Eductor Valve High Limit Switch
	ZSL_1301A				AT %I*					: BOOL;			// Eductor Valve Low Limit Switch
	HS_1301B				AT %Q*					: BOOL;			// Vacuum Diverter Valve
	ZSH_1301B				AT %I*					: BOOL;			// Vacuum Diverter Valve High Limit Switch
	ZSL_1301B				AT %I*					: BOOL;			// Vacuum Diverter Valve Low Limit Switch
	TI_1303					AT %I*					: INT;			// Vacuum Temperature
	TI_1303_Error			AT %I*					: BOOL;			// Vacuum Temperature Error
	bTI_1303_ErrActive								: BOOL;
	HS_1301					AT %Q*					: BOOL;			// Vacuum Pump
	TI_1304					AT %I*					: INT;			// Vacuum Pump Outlet Temperature
	TI_1304_Error			AT %I*					: BOOL;			// Vacuum Pump Outlet Temperature Error
	bTI_1304_ErrActive								: BOOL;
	LIC_1300				AT %I*					: INT;			// Vacuum Pump Discharge Separation Level
	HS_1300B				AT %Q*					: BOOL;			// Automated Drain Valve
	ZSH_1300				AT %I*					: BOOL;			// Automated Drain Valve High Limit Switch
	ZSL_1300				AT %I*					: BOOL;			// Automated Drain Valve Low Limit Switch
	HS_1300A				AT %Q*					: BOOL;			// Vacuum Cooling Pump/Seal Water Circulation Pump
	LSH_1300A				AT %I*					: BOOL;			// Seal Water Circulation Pump Level High Switch
	LSL_1300A				AT %I*					: BOOL;			// Seal Water Circulation Pump Level Low Switch
	FI_1300					AT %I*					: INT;			// Flow Meter
	TI_1302					AT %I*					: INT;			// Vacuum Cooler Input Temperature
	TI_1302_Error			AT %I*					: BOOL;			// Vacuum Cooler Input Temperature Error
	bTI_1302_ErrActive								: BOOL;
	HS_1305					AT %Q*					: BOOL;			// Vacuum Cooler Motor
	TI_1301					AT %I*					: INT;			// Vacuum Cooler Output Temperature
	TI_1301_Error			AT %I*					: BOOL;			// Vacuum Cooler Output Temperature Error
	bTI_1301_ErrActive								: BOOL;
	FI_1301					AT %I*					: INT;			// CO2 Product Flow
	AI_1301					AT %I*					: INT;			// CO2 Product Purity

	// Heat Traces
	TI_1					AT %I*					: INT;			// Heat Trace 1 Temperature
	TI_1_Error				AT %I*					: BOOL;			// Heat Trace 1 Temperature Error
	bTI_1_ErrActive									: BOOL;
	TI_2					AT %I*					: INT;			// Heat Trace 2 Temperature
	TI_2_Error				AT %I*					: BOOL;			// Heat Trace 2 Temperature Error
	bTI_2_ErrActive									: BOOL;
	TI_3					AT %I*					: INT;			// Heat Trace 3 Temperature
	TI_3_Error				AT %I*					: BOOL;			// Heat Trace 3 Temperature Error
	bTI_3_ErrActive									: BOOL;
	TI_4					AT %I*					: INT;			// Heat Trace 4 Temperature
	TI_4_Error				AT %I*					: BOOL;			// Heat Trace 4 Temperature Error
	bTI_4_ErrActive									: BOOL;
	TI_5					AT %I*					: INT;			// Heat Trace 5 Temperature
	TI_5_Error				AT %I*					: BOOL;			// Heat Trace 5 Temperature Error
	bTI_5_ErrActive									: BOOL;
	TI_6					AT %I*					: INT;			// Heat Trace 6 Temperature
	TI_6_Error				AT %I*					: BOOL;			// Heat Trace 6 Temperature Error
	bTI_6_ErrActive									: BOOL;
	TI_7					AT %I*					: INT;			// Heat Trace 7 Temperature
	TI_7_Error				AT %I*					: BOOL;			// Heat Trace 7 Temperature Error
	bTI_7_ErrActive									: BOOL;
	TI_8					AT %I*					: INT;			// Heat Trace 8 Temperature
	TI_8_Error				AT %I*					: BOOL;			// Heat Trace 8 Temperature Error
	bTI_8_ErrActive									: BOOL;
	TI_9					AT %I*					: INT;			// Heat Trace 9 Temperature
	TI_9_Error				AT %I*					: BOOL;			// Heat Trace 9 Temperature Error
	bTI_09_ErrActive								: BOOL;
	TI_10					AT %I*					: INT;			// Heat Trace 10 Temperature
	TI_10_Error				AT %I*					: BOOL;			// Heat Trace 10 Temperature Error
	bTI_10_ErrActive								: BOOL;
	TI_11					AT %I*					: INT;			// Heat Trace 11 Temperature
	TI_11_Error				AT %I*					: BOOL;			// Heat Trace 11 Temperature Error
	bTI_11_ErrActive								: BOOL;
	TI_12					AT %I*					: INT;			// Heat Trace 12 Temperature
	TI_12_Error				AT %I*					: BOOL;			// Heat Trace 12 Temperature Error
	bTI_12_ErrActive	 							: BOOL;
	HT_1_RELAY				AT %Q*					: BOOL;
	HT_2_RELAY				AT %Q*					: BOOL;
	HT_3_RELAY				AT %Q*					: BOOL;
	HT_4_RELAY				AT %Q*					: BOOL;
	HT_5_RELAY				AT %Q*					: BOOL;
	HT_6_RELAY				AT %Q*					: BOOL;
	HT_1_CTRL				AT %Q*					: INT;
	HT_2_CTRL				AT %Q*					: INT;
	HT_3_CTRL				AT %Q*					: INT;
	HT_4_CTRL				AT %Q*					: INT;
	HT_5_CTRL				AT %Q*					: INT;
	HT_6_CTRL				AT %Q*					: INT;
	
	HS_1102_Enable			AT %Q*					: BOOL;
	HS_1102_Out				AT %Q*					: INT;					
	
	// Current & Voltage measuement
	IT_1					AT %I*					: INT;
	IT_2					AT %I*					: INT;
	IT_3					AT %I*					: INT;
	VT_1					AT %I*					: INT;
	VT_2					AT %I*					: INT;
	VT_3					AT %I*					: INT;
	
	// LED Outputs
	LED1_R					AT %Q*					: BOOL;
	LED1_G					AT %Q*					: BOOL;
	LED1_Buzzer				AT %Q*					: BOOL;
	LED2_R					AT %Q*					: BOOL;
	LED2_G					AT %Q*					: BOOL;
	LED2_Buzzer				AT %Q*					: BOOL;

	// Lightbar                                 	
	LED3_R					AT %Q*					: BOOL;
	LED3_Y					AT %Q*					: BOOL;
	LED3_G					AT %Q*					: BOOL;
	LED3_Buzzer				AT %Q*					: BOOL;
	
	// Weather Station
	MI_2001					AT %I*					: INT;
	TI_2001					AT %I*					: INT;
	SI_2001					AT %I*					: INT;
	ZI_2001					AT %I*					: INT;
	PI_2001					AT %I*					: INT;
	
	// Inclinometer
	ZXI_2002				AT %I*					: WORD;
	ZYI_2002				AT %I*					: WORD;
	                                            	
	LightBar_Green			AT %Q*					: BOOL;
	Lightbar_Yellow			AT %Q*					: BOOL;
	Lightbar_Red			AT %Q*					: BOOL;
	                                            	
END_VAR

// ---- GVLs/Global_Variables_Tags.TcGVL
// Calvin - Global_Variables_Tags
// Rev 1.00 - September 20, 2023

VAR_GLOBAL
	
	// {attribute 'OPC.UA.DA.Access' := '3'}			// 1=Read Only, 2=Write Only, 3=Read/Write (Default)
	tgs_Current_User								: STRING;																// 7/21/23 PS - Added current user for HMI control
	{attribute 'OPC.UA.DA' := '3'}  				
	tgi_Current_User_Level							: INT;																	// 7/21/23 PS - Added current user level for HMI control
	{attribute 'OPC.UA.DA' := '3'}  				
	tgb_Hmi_Locked									: BOOL;																	// 7/22/23 PS - Added current user level for HMI control
	{attribute 'OPC.UA.DA' := '3'}  				
	tgs_Hmi_Log_Date_Time							: STRING;																// 7/22/23 PS - Added current user level for HMI control

	{attribute 'OPC.UA.DA' := '3'}  				
	tgr_SP_Adsorption_Time							: REAL;
	{attribute 'OPC.UA.DA' := '3'}  				                
	tgr_SP_Adsorption_CO2_Differential				: REAL;
	{attribute 'OPC.UA.DA' := '3'}  				
	tgr_SP_Adsorption_CO2_Time						: REAL;
	{attribute 'OPC.UA.DA' := '3'}
	tgr_SP_Boiler_Temp								: REAL;
	{attribute 'OPC.UA.DA' := '3'}
	tgr_SP_Boiler_Pressure							: REAL;
	{attribute 'OPC.UA.DA' := '3'}  				                
	tgr_SP_Min_LRP_Cooling_Loop_Flow				: REAL;
	{attribute 'OPC.UA.DA' := '3'}  				                
	tgr_SP_Evacuation_Target_Pressure				: REAL;
	{attribute 'OPC.UA.DA' := '3'}  				                
	tgr_SP_Evacuation_Target_Pressure_Steam			: REAL;																	// 07/14/23 PS - Added set point
	{attribute 'OPC.UA.DA' := '3'}  				                
	tgr_SP_Max_Allowed_Pressure_Leakage				: REAL;
	{attribute 'OPC.UA.DA' := '3'}
	tgr_SP_Reactor_Repressurization_Pressure		: REAL;
	{attribute 'OPC.UA.DA' := '3'}  				
	tgr_SP_Adsorption_Temp							: REAL;
	{attribute 'OPC.UA.DA' := '3'}  				                
	tgr_SP_Adsorption_VFD_Output					: REAL;
	{attribute 'OPC.UA.DA' := '3'}  				                
	tgr_SP_Min_Bypass_Steam_Flow					: REAL;
	{attribute 'OPC.UA.DA' := '3'}  				                
	tgr_SP_Min_Bypass_Steam_Temp					: REAL;
	{attribute 'OPC.UA.DA' := '3'}  				
	tgr_SP_IP_1302B_Reactor_Low						: REAL;
	{attribute 'OPC.UA.DA' := '3'}  				      
	tgr_SP_IP_1302B_Reactor_High					: REAL;
	{attribute 'OPC.UA.DA' := '3'}  				      
	tgr_SP_IP_1302B_Valve_Low						: REAL;
	{attribute 'OPC.UA.DA' := '3'}  				      
	tgr_SP_IP_1302B_Valve_High						: REAL;
	{attribute 'OPC.UA.DA' := '3'}  				      
	tgr_SP_Steam_Valve_Percent_Open					: REAL;
	{attribute 'OPC.UA.DA' := '3'}  				      
	tgr_SP_Max_Allowed_Sorbent_Temp					: REAL;
	{attribute 'OPC.UA.DA' := '3'}                        
	tgr_SP_Steam_Repressurization_Pressure			: REAL;
	{attribute 'OPC.UA.DA' := '3'}                        
	tgr_SP_Steam_Purge_Time							: REAL;
	{attribute 'OPC.UA.DA' := '3'}                        
	tgr_SP_Steam_Purge_Cutoff_Temp					: REAL;
	{attribute 'OPC.UA.DA' := '3'}                        
	tgr_SP_Evap_Cooling_Cutoff_Temp					: REAL;
	{attribute 'OPC.UA.DA' := '3'}                        
	tgr_SP_Evap_Cooling_Target_Pressure				: REAL;
	{attribute 'OPC.UA.DA' := '3'}                        
	tgr_SP_Leak_Check_Time							: REAL;
	
	{attribute 'OPC.UA.DA' := '3'}  				                
	tgb_Warmup_Complete								: BOOL;
	{attribute 'OPC.UA.DA' := '3'}  				                
	tgb_HMI_Active									: BOOL;						// An HMI program is running and communicating
	{attribute 'OPC.UA.DA' := '2'}  				                
	tgb_Auto_Mode									: BOOL;						// Machine is in Auto Mode
	{attribute 'OPC.UA.DA' := '1'}  				                
	tgb_Watchdog									: BOOL;
	{attribute 'OPC.UA.DA' := '1'}  				                
	tgb_ADS_Active									: BOOL;						// ADS HMI program is running and communicating
	{attribute 'OPC.UA.DA' := '1'}  				
	tgb_Active_Alarm								: BOOL;
	{attribute 'OPC.UA.DA' := '3'}  				                
	tgb_Alarm_Reset									: BOOL;
	{attribute 'OPC.UA.DA' := '1'}  				
	tgb_Half_Sec_Pulse								: BOOL;
	{attribute 'OPC.UA.DA' := '3'}  				
	tgb_File_Save_Error								: BOOL;
	{attribute 'OPC.UA.DA' := '3'}  				                
	tgb_Test_Mode									: BOOL;						// Start or stop test
	{attribute 'OPC.UA.DA' := '1'}  				                
	tgb_Test_Running								: BOOL;						// Test is running
	{attribute 'OPC.UA.DA' := '1'}  				
	tgb_Stop_Cycle									: BOOL;
	{attribute 'OPC.UA.DA' := '1'}  				
	tgi_Current_Step								: INT;
	{attribute 'OPC.UA.DA' := '1'}  				
	tgi_Machine_State								: INT;
	{attribute 'OPC.UA.DA' := '1'}  				
	tgi_Alarm_State									: INT;						// Current Alarm State
	{attribute 'OPC.UA.DA' := '1'}  				
	tgi_Cycles_To_Run								: INT;
	{attribute 'OPC.UA.DA' := '1'}  				
	tgi_Cycle_Count									: INT;						// Number of TVSA cycles run since cycle restart
	{attribute 'OPC.UA.DA' := '1'}  				
	tgi_Status										: INT;
	{attribute 'OPC.UA.DA' := '1'}  				
	tgi_Total_Cycle_Count							: DINT;						// Total number of TVSA cycles run
	{attribute 'OPC.UA.DA' := '1'}  				
	tgr_Remaining_Time								: REAL;
	{attribute 'OPC.UA.DA' := '1'}  				
	tgs_Alarm										: STRING;
	{attribute 'OPC.UA.DA' := '1'}  				
	tgs_Active_Alarm								: STRING;
	{attribute 'OPC.UA.DA' := '1'}  				
	tgs_Status										: STRING;
	
	{attribute 'OPC.UA.DA' := '3'}  				
	tgb_Drains_On									: BOOL;
	{attribute 'OPC.UA.DA' := '3'}  				                
	tgb_Manual_Heater_Mode							: BOOL;						// Manual heater mode active
	{attribute 'OPC.UA.DA' := '1'}  				
	tgb_Adsorption_CO2								: BOOL;

	
	// Reactor
	{attribute 'OPC.UA.DA' := '1'}  				                
	tgr_DPT_1102A									: REAL;			
	{attribute 'OPC.UA.DA' := '1'}  				                
	tgr_FIC_1102									: REAL;			
	{attribute 'OPC.UA.DA' := '1'}  				                
	tgr_AI_1102A									: REAL;			
	{attribute 'OPC.UA.DA' := '3'}  				                
	tgb_AI_1102A_Pump								: BOOL;			
	{attribute 'OPC.UA.DA' := '1'}  				                
	tgb_AI_1102A_Pump_On							: BOOL;			
	{attribute 'OPC.UA.DA' := '3'}  				                
	tgb_AI_1102A_Solenoid							: BOOL;			
	{attribute 'OPC.UA.DA' := '1'}  				                
	tgb_AI_1102A_Solenoid_On						: BOOL;			
	{attribute 'OPC.UA.DA' := '1'}  				                
	tgr_MI_1102A									: REAL;			
	{attribute 'OPC.UA.DA' := '3'}  				                
	tgr_IP_1102A									: REAL;			
	{attribute 'OPC.UA.DA' := '3'}  				                
	tgr_IP_1102A_Output								: REAL;			
	{attribute 'OPC.UA.DA' := '1'}  				                
	tgr_ZT_1102A									: REAL;			
	{attribute 'OPC.UA.DA' := '1'}  				                
	tgr_PI_1100										: REAL;			
	{attribute 'OPC.UA.DA' := '1'}  				                
	tgr_DPT_1100									: REAL;			
	{attribute 'OPC.UA.DA' := '3'}  				                
	tgr_IP_1102B									: REAL;			
	{attribute 'OPC.UA.DA' := '3'}  				                
	tgr_IP_1102B_Output								: REAL;			
	{attribute 'OPC.UA.DA' := '1'}  				                
	tgr_ZT_1102B									: REAL;			
	{attribute 'OPC.UA.DA' := '1'}  				                
	tgr_AI_1102B									: REAL;			
	{attribute 'OPC.UA.DA' := '3'}  				                
	tgb_AI_1102B_Pump								: BOOL;			
	{attribute 'OPC.UA.DA' := '1'}  				                
	tgb_AI_1102B_Pump_On							: BOOL;			
	{attribute 'OPC.UA.DA' := '3'}  				                
	tgb_AI_1102B_Solenoid							: BOOL;			
	{attribute 'OPC.UA.DA' := '1'}  				                
	tgb_AI_1102B_Solenoid_On						: BOOL;			
	{attribute 'OPC.UA.DA' := '1'}  				                
	tgr_MI_1102B									: REAL;			
	{attribute 'OPC.UA.DA' := '1'}  				                
	tgr_DPT_1102B									: REAL;			
	{attribute 'OPC.UA.DA' := '1'}  				                
	tgr_TI_1102A									: REAL;			
	{attribute 'OPC.UA.DA' := '1'}  				                
	tgb_TI_1102A_Error								: BOOL;			
	{attribute 'OPC.UA.DA' := '1'}  				                
	tgr_TI_1100A									: REAL;			
	{attribute 'OPC.UA.DA' := '1'}  				                
	tgb_TI_1100A_Error								: BOOL;			
	{attribute 'OPC.UA.DA' := '1'}  				                
	tgr_TI_1100B									: REAL;			
	{attribute 'OPC.UA.DA' := '1'}  				                
	tgb_TI_1100B_Error								: BOOL;			
	{attribute 'OPC.UA.DA' := '1'}  				                
	tgr_TI_1100C									: REAL;			
	{attribute 'OPC.UA.DA' := '1'}  				                
	tgb_TI_1100C_Error								: BOOL;			
	{attribute 'OPC.UA.DA' := '1'}  				                
	tgr_TI_1102B									: REAL;			
	{attribute 'OPC.UA.DA' := '1'}  				                
	tgb_TI_1102B_Error								: BOOL;			

	{attribute 'OPC.UA.DA' := '3'}  				                
	tgr_HS_1102									: REAL;
	{attribute 'OPC.UA.DA' := '3'}  				                
	tgr_HS_1102_Output								: REAL;
	{attribute 'OPC.UA.DA' := '1'}  				                
	tgr_HS_1102_RPM									: REAL;			// Fan rpm
	{attribute 'OPC.UA.DA' := '1'}  				                
	tgr_HS_1102V									: REAL;			// VFD frequency
	{attribute 'OPC.UA.DA' := '1'}  				                
	tgb_HS_1102_Enabled								: BOOL;			// VFD enabled	
	{attribute 'OPC.UA.DA' := '1'}  				                
	tgb_HS_1102_Running								: BOOL;			// Fan running
	{attribute 'OPC.UA.DA' := '1'}  				                
	tgb_HS_1104										: BOOL;			
	{attribute 'OPC.UA.DA' := '1'}  				                
	tgb_HS_1104_On									: BOOL;			
	{attribute 'OPC.UA.DA' := '1'}  				                
	tgb_HS_1104_Open								: BOOL;			
	{attribute 'OPC.UA.DA' := '1'}  				                
	tgb_HS_1104_Closed								: BOOL;			
	
	{attribute 'OPC.UA.DA' := '1'}  				                
	tgb_IP_1102A_Open								: BOOL;			
	{attribute 'OPC.UA.DA' := '1'}  				                
	tgb_IP_1102A_Closed								: BOOL;			
	{attribute 'OPC.UA.DA' := '1'}  				                
	tgb_IP_1102B_Open								: BOOL;			
	{attribute 'OPC.UA.DA' := '1'}  				                
	tgb_IP_1102B_Closed								: BOOL;			
	{attribute 'OPC.UA.DA' := '3'}  				                
	tgb_YL_1001										: BOOL;			
	{attribute 'OPC.UA.DA' := '1'}  				                
	tgb_YL_1001_On									: BOOL;			

	{attribute 'OPC.UA.DA' := '1'}  				                
	tgr_FI_1200_1									: REAL;			
	{attribute 'OPC.UA.DA' := '1'}  				                
	tgr_FI_1200_2									: REAL;			
	{attribute 'OPC.UA.DA' := '1'}  				                
	tgr_FI_1200_3									: REAL;			
	{attribute 'OPC.UA.DA' := '1'}  				                
	tgr_FI_1201_1									: REAL;			
	{attribute 'OPC.UA.DA' := '1'}  				                
	tgr_FI_1201_2									: REAL;			
	{attribute 'OPC.UA.DA' := '1'}  				                
	tgr_FI_1201_3									: REAL;			
	{attribute 'OPC.UA.DA' := '1'}  				                
	tgr_PI_1200										: REAL;			
	{attribute 'OPC.UA.DA' := '1'}  				                
	tgr_PI_1001										: REAL;			
	{attribute 'OPC.UA.DA' := '1'}  				                
	tgr_TI_1001										: REAL;			
	{attribute 'OPC.UA.DA' := '1'}  				                
	tgb_TI_1001_Error								: BOOL;			
	{attribute 'OPC.UA.DA' := '1'}  				                
	tgr_FI_1001										: REAL;			
	{attribute 'OPC.UA.DA' := '3'}  				                
	tgr_IP_1101										: REAL;			
	{attribute 'OPC.UA.DA' := '3'}  				                
	tgr_IP_1101_Output								: REAL;			
	{attribute 'OPC.UA.DA' := '1'}  				                
	tgr_ZT_1101										: REAL;			
	{attribute 'OPC.UA.DA' := '1'}  				                
	tgr_PI_1101										: REAL;			
	{attribute 'OPC.UA.DA' := '1'}  				                
	tgr_TI_1101										: REAL;			
	{attribute 'OPC.UA.DA' := '1'}  				                
	tgb_TI_1101_Error								: BOOL;			
	{attribute 'OPC.UA.DA' := '3'}  				                
	tgb_HS_1107										: BOOL;			
	{attribute 'OPC.UA.DA' := '1'}  				                
	tgb_HS_1107_On									: BOOL;			
	{attribute 'OPC.UA.DA' := '1'}  				                
	tgb_HS_1107_Open								: BOOL;			
	{attribute 'OPC.UA.DA' := '1'}  				                
	tgb_HS_1107_Closed								: BOOL;			
	{attribute 'OPC.UA.DA' := '3'}  				                
	tgb_HS_1101A									: BOOL;			
	{attribute 'OPC.UA.DA' := '1'}  				                
	tgb_HS_1101A_On									: BOOL;			
	{attribute 'OPC.UA.DA' := '1'}  				                
	tgb_HS_1101A_Open								: BOOL;			
	{attribute 'OPC.UA.DA' := '1'}  				                
	tgb_HS_1101A_Closed								: BOOL;			
	{attribute 'OPC.UA.DA' := '3'}  				                
	tgb_HS_1101B									: BOOL;			
	{attribute 'OPC.UA.DA' := '1'}  				                
	tgb_HS_1101B_On									: BOOL;			
	{attribute 'OPC.UA.DA' := '1'}  				                
	tgb_HS_1101B_Open								: BOOL;			
	{attribute 'OPC.UA.DA' := '1'}  				                
	tgb_HS_1101B_Closed								: BOOL;			
	{attribute 'OPC.UA.DA' := '1'}  				                
	tgr_TI_1103										: REAL;			
	{attribute 'OPC.UA.DA' := '1'}  				                
	tgb_TI_1103_Error								: BOOL;			
	{attribute 'OPC.UA.DA' := '1'}  				                
	tgr_TI_1104										: REAL;			
	{attribute 'OPC.UA.DA' := '1'}  				                
	tgb_TI_1104_Error								: BOOL;			
	{attribute 'OPC.UA.DA' := '1'}  				                
	tgr_TI_1105										: REAL;			
	{attribute 'OPC.UA.DA' := '1'}  				                
	tgb_TI_1105_Error								: BOOL;			
	{attribute 'OPC.UA.DA' := '1'}  				                
	tgr_TI_1106										: REAL;			
	{attribute 'OPC.UA.DA' := '1'}  				                
	tgb_TI_1106_Error								: BOOL;			

	// Condensate
	{attribute 'OPC.UA.DA' := '3'}  				                
	tgb_HS_1201										: BOOL;			
	{attribute 'OPC.UA.DA' := '1'}  				                
	tgb_HS_1201_On									: BOOL;			
	{attribute 'OPC.UA.DA' := '1'}  				                
	tgb_HS_1201_LSH									: BOOL;			
	{attribute 'OPC.UA.DA' := '1'}  				                
	tgb_HS_1201_LSL									: BOOL;			
	{attribute 'OPC.UA.DA' := '3'}  				                
	tgb_HS_1103A									: BOOL;			
	{attribute 'OPC.UA.DA' := '1'}  				                
	tgb_HS_1103A_On									: BOOL;			
	{attribute 'OPC.UA.DA' := '1'}  				                
	tgb_HS_1103A_Open								: BOOL;			
	{attribute 'OPC.UA.DA' := '1'}  				                
	tgb_HS_1103A_Closed								: BOOL;			
	{attribute 'OPC.UA.DA' := '3'}  				                
	tgr_IP_1302B									: REAL;			
	{attribute 'OPC.UA.DA' := '3'}  				                
	tgr_IP_1302B_Output								: REAL;			
	{attribute 'OPC.UA.DA' := '1'}  				                
	tgr_ZT_1302B									: REAL;			
	{attribute 'OPC.UA.DA' := '3'}  				                
	tgb_HS_1103B									: BOOL;			
	{attribute 'OPC.UA.DA' := '1'}  				                
	tgb_HS_1103B_On									: BOOL;			
	{attribute 'OPC.UA.DA' := '1'}  				                
	tgb_HS_1103B_Open								: BOOL;			
	{attribute 'OPC.UA.DA' := '1'}  				                
	tgb_HS_1103B_Closed								: BOOL;			
	{attribute 'OPC.UA.DA' := '3'}  				                
	tgb_HS_1203										: BOOL;			
	{attribute 'OPC.UA.DA' := '3'}  				                
	tgb_HS_1203_On									: BOOL;			
	{attribute 'OPC.UA.DA' := '3'}  				                
	tgb_HS_1202										: BOOL;			
	{attribute 'OPC.UA.DA' := '1'}  				                
	tgb_HS_1202_On									: BOOL;			
	{attribute 'OPC.UA.DA' := '1'}  				                
	tgb_HS_1202_LSH									: BOOL;			
	{attribute 'OPC.UA.DA' := '1'}  				                
	tgb_HS_1202_LSL									: BOOL;			
	{attribute 'OPC.UA.DA' := '1'}  				                
	tgr_LI_1204										: REAL;			
	{attribute 'OPC.UA.DA' := '3'}  				                
	tgb_HS_1200										: BOOL;			
	{attribute 'OPC.UA.DA' := '1'}  				                
	tgb_HS_1200_On									: BOOL;			
	{attribute 'OPC.UA.DA' := '3'}  				                
	tgb_SV_1201										: BOOL;			
	{attribute 'OPC.UA.DA' := '1'}  				                
	tgb_SV_1201_On									: BOOL;			
	{attribute 'OPC.UA.DA' := '1'}  				                
	tgb_SV_1201_Open								: BOOL;			
	{attribute 'OPC.UA.DA' := '1'}  				                
	tgb_SV_1201_Closed								: BOOL;			
	
	// Vacuum
	{attribute 'OPC.UA.DA' := '1'}  				                
	tgr_AI_1300_1									: REAL;			
	{attribute 'OPC.UA.DA' := '1'}  				                
	tgr_AI_1300_2									: REAL;			
	{attribute 'OPC.UA.DA' := '1'}  				                
	tgr_AI_1300_3									: REAL;			
	{attribute 'OPC.UA.DA' := '3'}  				                
	tgb_HS_1302A									: BOOL;			
	{attribute 'OPC.UA.DA' := '1'}  				                
	tgb_HS_1302A_On									: BOOL;			
	{attribute 'OPC.UA.DA' := '1'}  				                
	tgb_HS_1302A_Open								: BOOL;			
	{attribute 'OPC.UA.DA' := '1'}  				                
	tgb_HS_1302A_Closed								: BOOL;			
	{attribute 'OPC.UA.DA' := '1'}  				                
	tgr_PI_1300										: REAL;			
	{attribute 'OPC.UA.DA' := '3'}  				                
	tgb_HS_1301A									: BOOL;			
	{attribute 'OPC.UA.DA' := '1'}  				                
	tgb_HS_1301A_On									: BOOL;			
	{attribute 'OPC.UA.DA' := '1'}  				                
	tgb_HS_1301A_Open								: BOOL;			
	{attribute 'OPC.UA.DA' := '1'}  				                
	tgb_HS_1301A_Closed								: BOOL;			
	{attribute 'OPC.UA.DA' := '3'}  				                
	tgb_HS_1301B									: BOOL;			
	{attribute 'OPC.UA.DA' := '1'}  				                
	tgb_HS_1301B_On									: BOOL;			
	{attribute 'OPC.UA.DA' := '1'}  				                
	tgb_HS_1301B_Open								: BOOL;			
	{attribute 'OPC.UA.DA' := '1'}  				                
	tgb_HS_1301B_Closed								: BOOL;			
	{attribute 'OPC.UA.DA' := '1'}  				                
	tgr_TI_1303										: REAL;			
	{attribute 'OPC.UA.DA' := '1'}  				                
	tgb_TI_1303_Error								: BOOL;
	{attribute 'OPC.UA.DA' := '3'}  				                
	tgb_HS_1301										: BOOL;			
	{attribute 'OPC.UA.DA' := '1'}  				                
	tgb_HS_1301_On									: BOOL;			
	{attribute 'OPC.UA.DA' := '1'}  				                
	tgr_TI_1304										: REAL;			
	{attribute 'OPC.UA.DA' := '1'}  				                
	tgb_TI_1304_Error								: BOOL;
	{attribute 'OPC.UA.DA' := '1'}  				                
	tgr_LIC_1300									: REAL;			
	{attribute 'OPC.UA.DA' := '3'}  				                
	tgb_HS_1300B									: BOOL;
	{attribute 'OPC.UA.DA' := '1'}  				                
	tgb_HS_1300B_On									: BOOL;
	{attribute 'OPC.UA.DA' := '1'}  				                
	tgb_HS_1300B_Open								: BOOL;			
	{attribute 'OPC.UA.DA' := '1'}  				                
	tgb_HS_1300B_Closed								: BOOL;			
	{attribute 'OPC.UA.DA' := '3'}  				                
	tgb_HS_1300A									: BOOL;			
	{attribute 'OPC.UA.DA' := '1'}  				                
	tgb_HS_1300A_On									: BOOL;			
	{attribute 'OPC.UA.DA' := '1'}  				                
	tgb_HS_1300A_LSH								: BOOL;			
	{attribute 'OPC.UA.DA' := '1'}  				                
	tgb_HS_1300A_LSL								: BOOL;			
	{attribute 'OPC.UA.DA' := '1'}  				                
	tgr_FI_1300										: REAL;			
	{attribute 'OPC.UA.DA' := '1'}  				                
	tgr_TI_1302										: REAL;			
	{attribute 'OPC.UA.DA' := '1'}  				                
	tgb_TI_1302_Error								: BOOL;			
	{attribute 'OPC.UA.DA' := '3'}  				                
	tgb_HS_1305										: BOOL;			
	{attribute 'OPC.UA.DA' := '1'}  				                
	tgb_HS_1305_On									: BOOL;			
	{attribute 'OPC.UA.DA' := '1'}  				                
	tgr_TI_1301										: REAL;			
	{attribute 'OPC.UA.DA' := '1'}  				                
	tgb_TI_1301_Error								: BOOL;			
	{attribute 'OPC.UA.DA' := '1'}  				                
	tgr_FI_1301										: REAL;			
	{attribute 'OPC.UA.DA' := '1'}  				                
	tgr_AI_1301										: REAL;			
				                                           
	// Heat Traces
	{attribute 'OPC.UA.DA' := '3'}  				                
	tgr_HT_P_Value									: REAL;						// Trace heater P factor
	{attribute 'OPC.UA.DA' := '3'}  				                
	tgr_HT_I_Value									: REAL;						// Trace heater I factor
	{attribute 'OPC.UA.DA' := '3'}  				                
	tgr_HT_I_Range									: REAL;						// Plus-minus range that Integral value is active in PID loop
	{attribute 'OPC.UA.DA' := '3'}  				                
	tgi_Manual_Heater_Output						: INT	:= 0;				// Manual heater output value
	{attribute 'OPC.UA.DA' := '1'}  				                
	tgr_TI_1										: REAL;			
	{attribute 'OPC.UA.DA' := '1'}  				                
	tgb_TI_1_Error									: BOOL;			
	{attribute 'OPC.UA.DA' := '3'}  				                
	tgb_HT_1_On										: BOOL;			
	{attribute 'OPC.UA.DA' := '3'}  				                
	tgr_HT_1_SP										: REAL;			
	{attribute 'OPC.UA.DA' := '1'}  				                
	tgr_HT_1_Ctrl									: REAL;			
	{attribute 'OPC.UA.DA' := '3'}  				                
	tgr_HT_1_Manual_Output							: REAL;			
	{attribute 'OPC.UA.DA' := '3'}  				                
	tgr_HT_1_Base_Output							: REAL;			
	{attribute 'OPC.UA.DA' := '1'}  				                
	tgr_TI_2										: REAL;			
	{attribute 'OPC.UA.DA' := '1'}  				                
	tgb_TI_2_Error									: BOOL;			
	{attribute 'OPC.UA.DA' := '3'}  				                
	tgb_HT_2_On										: BOOL;			
	{attribute 'OPC.UA.DA' := '3'}  				                
	tgr_HT_2_SP										: REAL;			
	{attribute 'OPC.UA.DA' := '1'}  				                
	tgr_HT_2_Ctrl									: REAL;			
	{attribute 'OPC.UA.DA' := '3'}  				                
	tgr_HT_2_Manual_Output							: REAL;			
	{attribute 'OPC.UA.DA' := '3'}  				                
	tgr_HT_2_Base_Output							: REAL;			
	{attribute 'OPC.UA.DA' := '1'}  				                
	tgr_TI_3										: REAL;			
	{attribute 'OPC.UA.DA' := '1'}  				                
	tgb_TI_3_Error									: BOOL;			
	{attribute 'OPC.UA.DA' := '3'}  				                
	tgb_HT_3_On										: BOOL;			
	{attribute 'OPC.UA.DA' := '3'}  				                
	tgr_HT_3_SP										: REAL;			
	{attribute 'OPC.UA.DA' := '1'}  				                
	tgr_HT_3_Ctrl									: REAL;			
	{attribute 'OPC.UA.DA' := '3'}  				                
	tgr_HT_3_Manual_Output							: REAL;			
	{attribute 'OPC.UA.DA' := '3'}  				                
	tgr_HT_3_Base_Output							: REAL;			
	{attribute 'OPC.UA.DA' := '1'}  				                
	tgr_TI_4										: REAL;			
	{attribute 'OPC.UA.DA' := '1'}  				                
	tgb_TI_4_Error									: BOOL;			
	{attribute 'OPC.UA.DA' := '3'}  				                
	tgb_HT_4_On										: BOOL;			
	{attribute 'OPC.UA.DA' := '3'}  				                
	tgr_HT_4_SP										: REAL;			
	{attribute 'OPC.UA.DA' := '1'}  				                
	tgr_HT_4_Ctrl									: REAL;			
	{attribute 'OPC.UA.DA' := '3'}  				                
	tgr_HT_4_Manual_Output							: REAL;			
	{attribute 'OPC.UA.DA' := '3'}  				                
	tgr_HT_4_Base_Output							: REAL;			
	{attribute 'OPC.UA.DA' := '1'}  				                
	tgr_TI_5										: REAL;			
	{attribute 'OPC.UA.DA' := '1'}  				                
	tgb_TI_5_Error									: BOOL;			
	{attribute 'OPC.UA.DA' := '3'}  				                
	tgb_HT_5_On										: BOOL;			
	{attribute 'OPC.UA.DA' := '3'}  				                
	tgr_HT_5_SP										: REAL;			
	{attribute 'OPC.UA.DA' := '1'}  				                
	tgr_HT_5_Ctrl									: REAL;			
	{attribute 'OPC.UA.DA' := '3'}  				                
	tgr_HT_5_Manual_Output							: REAL;			
	{attribute 'OPC.UA.DA' := '3'}  				                
	tgr_HT_5_Base_Output							: REAL;			
	{attribute 'OPC.UA.DA' := '1'}  				                
	tgr_TI_6										: REAL;			
	{attribute 'OPC.UA.DA' := '1'}  				                
	tgb_TI_6_Error									: BOOL;			
	{attribute 'OPC.UA.DA' := '3'}  				                
	tgb_HT_6_On										: BOOL;			
	{attribute 'OPC.UA.DA' := '3'}  				                
	tgr_HT_6_SP										: REAL;			
	{attribute 'OPC.UA.DA' := '1'}  				                
	tgr_HT_6_Ctrl									: REAL;			
	{attribute 'OPC.UA.DA' := '3'}  				                
	tgr_HT_6_Manual_Output							: REAL;			
	{attribute 'OPC.UA.DA' := '3'}  				                
	tgr_HT_6_Base_Output							: REAL;			
	{attribute 'OPC.UA.DA' := '1'}  				                
	tgr_TI_7										: REAL;			
	{attribute 'OPC.UA.DA' := '1'}  				                
	tgb_TI_7_Error									: BOOL;			
	{attribute 'OPC.UA.DA' := '1'}  				                
	tgr_TI_8										: REAL;			
	{attribute 'OPC.UA.DA' := '1'}  				                
	tgb_TI_8_Error									: BOOL;			
	{attribute 'OPC.UA.DA' := '1'}  				                
	tgr_TI_9										: REAL;			
	{attribute 'OPC.UA.DA' := '1'}  				                
	tgb_TI_9_Error									: BOOL;			
	{attribute 'OPC.UA.DA' := '1'}  				                
	tgr_TI_10										: REAL;			
	{attribute 'OPC.UA.DA' := '1'}  				                
	tgb_TI_10_Error									: BOOL;			
	{attribute 'OPC.UA.DA' := '1'}  				                
	tgr_TI_11										: REAL;			
	{attribute 'OPC.UA.DA' := '1'}  				                
	tgb_TI_11_Error									: BOOL;			
	{attribute 'OPC.UA.DA' := '1'}  				                
	tgr_TI_12										: REAL;			
	{attribute 'OPC.UA.DA' := '1'}  				                
	tgb_TI_12_Error									: BOOL;			
	
	// Current & Voltage
	{attribute 'OPC.UA.DA' := '1'}  				                
	tgr_IT_1										: REAL;			
	{attribute 'OPC.UA.DA' := '1'}  				                
	tgr_IT_2										: REAL;			
	{attribute 'OPC.UA.DA' := '1'}  				                
	tgr_IT_3										: REAL;			
	{attribute 'OPC.UA.DA' := '1'}  				                
	tgr_VT_1										: REAL;			
	{attribute 'OPC.UA.DA' := '1'}  				                
	tgr_VT_2										: REAL;			
	{attribute 'OPC.UA.DA' := '1'}  				                
	tgr_VT_3										: REAL;			
	
	
	// Weather Station
	{attribute 'OPC.UA.DA' := '1'}  				                
	tgr_MI_2001										: REAL;			
	{attribute 'OPC.UA.DA' := '1'}  				                
	tgr_TI_2001										: REAL;			
	{attribute 'OPC.UA.DA' := '1'}  				                
	tgr_SI_2001										: REAL;			
	{attribute 'OPC.UA.DA' := '1'}  				                
	tgr_ZI_2001										: REAL;			
	{attribute 'OPC.UA.DA' := '1'}  				                
	tgr_PI_2001										: REAL;			

	// Inclinometer  				                
	{attribute 'OPC.UA.DA' := '1'}
	tgr_ZXI_2002									: REAL;			
	{attribute 'OPC.UA.DA' := '1'}  				                
	tgr_ZYI_2002									: REAL;			
	
END_VAR

// ---- POUs/MAIN.TcPOU
PROGRAM MAIN

VAR
	rtrigHmiStartup									: R_TRIG;
	ftrigHmiShutdown								: F_TRIG;
	tonHalfSecPulse									: TON;
	tonWatchdog										: TON;
	bMBWeather										: BOOL;
	iVFDCount										: INT;
END_VAR

// Calvin - MAIN
// Rev 1.00 - August 5, 2023

P_State_Machine();
P_AlarmCheck();
P_HeaterControl();
P_VFD_Test();

rtrigHmiStartup(CLK:= tgb_ADS_Active);
IF rtrigHmiStartup.Q THEN
//	gbRunVFD										:= TRUE;
	tgr_HS_1102										:= 0;
END_IF
ftrigHmiShutdown(CLK:= tgb_ADS_Active);
IF ftrigHmiShutdown.Q THEN
//	gbRunVFD										:= FALSE;
	eState											:= eReset;
	P_State_Machine.A0_Reset();
END_IF

/// TIMER PULSE
IF tonHalfSecPulse.Q THEN
	tgb_Half_Sec_Pulse								:= NOT tgb_Half_Sec_Pulse;
	tgb_Watchdog									:= TRUE;
	tonHalfSecPulse(IN:= FALSE);
	iVFDCount										:= iVFDCount + 1;
	IF iVFDCount >= 4 THEN
		iVFDCount									:= 0;
		gbReadMBVFD									:= TRUE;
		IF bMBWeather THEN
			gbReadMBWeather							:= TRUE;
		ELSE
			gbReadMBInclinometer					:= TRUE;
		END_IF
		bMBWeather									:= NOT bMBWeather;
	END_IF
END_IF
tonHalfSecPulse(IN:= TRUE, PT:= T#500MS);

(*IF tonWatchdog.Q THEN
	tgb_ADS_Active									:= FALSE;
END_IF
tonWatchdog(IN:= tgb_Watchdog AND tgb_ADS_Active, PT:= T#4S);	*)

END_PROGRAM

// ---- POUs/P_State_Machine.TcPOU
PROGRAM P_State_Machine
VAR RETAIN
	gpdiCycle_Count									: DINT;
END_VAR
VAR
	strStatusLabel									: ARRAY[0..50] OF STRING;
	strError										: STRING;
	strProcessError									: STRING;
	bStatusListLoaded								: BOOL;	
	
	rtrigWarmup										: R_TRIG;
	rtrigEvacuation									: R_TRIG;
	rtrigSteamBypass								: R_TRIG;
	rtrigDesorption									: R_TRIG;
	rtrigRepressurization							: R_TRIG;
	rtrigAdsorption									: R_TRIG;
	rtrigStatusReady								: R_TRIG;

	iStep											: INT;
	i1Step											: INT;
	i2Step											: INT;
	i3Step											: INT;
	i4Step											: INT;
	i5Step											: INT;
	i6Step											: INT;
	
	bVacuumHolding									: BOOL;
	bWarmUpDone										: BOOL;
	bRunEvacuation									: BOOL;
	bEvacuationDone									: BOOL;
	bSteamBypassDone								: BOOL;
	bDesorptionDone							        : BOOL;
	bRepressurizationDone							: BOOL;
	bAdsorptionDone									: BOOL;
	bRunning										: BOOL;
	bInRange1										: BOOL;
	bInRange2										: BOOL;
	bInRange3										: BOOL;
	bTempAGood										: BOOL;
	bTempBGood										: BOOL;
	bTempCGood										: BOOL;
	bOverTemp										: BOOL;
	bStop											: BOOL;
	bTimer1											: BOOL;
	bTimer2											: BOOL;
	rTime1											: REAL;
	rTime2											: REAL;
	rSP1											: REAL;
	rSP2											: REAL;
	tonTimer1										: TON;
	tonTimer2										: TON;
	tonReset										: TON;
	tonPause										: TON;

	bRunValveModulation								: BOOL;
	bValveInRange									: BOOL;
	bFanError										: BOOL;
	bClearDrains									: BOOL;
	bCondenserLow									: BOOL;				// 09/07/23 PS
	bCondenserFull									: BOOL;				// 09/19/23 PS
	bCondenserRefill								: BOOL;				// 09/21/23 PS
	rOut											: REAL;
	rPI_1100_Save									: REAL;
	
	bDrainLSHClear									: BOOL;
	bDrainLSLClear									: BOOL;
	b1200DrainOROff									: BOOL;				// AF_Drains 4/7/23
	b1201DrainOn									: BOOL;				// AF_Drains 4/7/23
	b1202DrainOn									: BOOL;				// AF_Drains 4/7/23
	b1300DrainOn									: BOOL;				// 09/21/23 PS
	bDrainOn										: BOOL;				// AF_Drains 4/7/23
	b1201DrainOROff									: BOOL;				// 09/20/23 PS
	b1202DrainOROff									: BOOL;				// 09/20/23 PS
	b1202DrainOROn									: BOOL;				// 09/20/23 PS
	rtrigDrainsOff									: R_TRIG;			// 09/20/23 PS
	
	// A_DPT_Fan_Test
	tonFanTest										: TON;
	rtrigFanTest									: R_TRIG;
	ftrigFanTest									: F_TRIG;	
	tFanTestTime									: TIME	:= T#60S;
	rHS_1102										: REAL	:= 0.0;
	rFanIncrement									: REAL	:= 10.0;
	rFanMaximum										: REAL	:= 100.0;
	iFanTestStep									: INT	:= 0;
	bFanTimer										: BOOL;

	// A_Modbus_VFD
	MBV_Master 										: ModbusRtuMasterV2_KL6x22B;	
	MBV_Errors										: MODBUS_ERRORS;
	tonMBVReset										: TON;
	bMBVBusy										: BOOL;
	bMBVError										: BOOL;
	bMBVReadStatus									: BOOL;
	bMBVStatusCheck									: BOOL;
	iMBVFunction									: INT;
	iMBVHzRetry										: INT;
	uiMBVRead										: UINT;	
	wMBVAddress										: WORD;
	wMBVQuantity									: WORD;
	wMBVOnOff										: WORD;
	wMBVStatus										: WORD 	:= 3;
	wMBVReadData 									: ARRAY[0..21] OF WORD;
	wMBVWriteData 									: ARRAY[0..21] OF WORD;
	// A_Modbus_Points
	MBP_Master 										: ModbusRtuMasterV2_KL6x22B;	
	MBP_Errors										: MODBUS_ERRORS;
	tonMBPReset										: TON;
	bMBPWeather										: BOOL;
	bMBPBusy										: BOOL;
	bMBPError										: BOOL;
	iMBPFunction									: INT;
	uiMBPRead										: UINT;	
	wMBPAddress										: WORD;
	wMBPQuantity									: WORD;
	wMBPReadData 									: ARRAY[0..21] OF WORD;
	wMBPWriteData 									: ARRAY[0..21] OF WORD;

END_VAR

// Calvin - P_State_Machine
// Rev 1.00 - September 21, 2023

IF NOT bStatusListLoaded THEN
	A_Status_List();
END_IF

A_Temperatures();																											// Run these actions continuously
A_Inputs_Outputs();
A_Interlocks();
A_Modbus_VFD();
//A_Modbus_Points();
A_DPT_Fan_Test();
A_WaterHandling();

rtrigWarmup(CLK:= tgi_Machine_State = eWarmup);																				// Set trigger (one shot) on initial entry of each state
rtrigEvacuation(CLK:= tgi_Machine_State = eEvacuation);
rtrigSteamBypass(CLK:= tgi_Machine_State = eSteamBypass);
rtrigDesorption(CLK:= tgi_Machine_State = eDesorption);
rtrigRepressurization(CLK:= tgi_Machine_State = eRepressurization);
rtrigAdsorption(CLK:= tgi_Machine_State = eAdsorption);

IF rtrigWarmup.Q THEN																										// Warm up triggered
	bWarmUpDone										:= FALSE;																// Clear Done flag
	i1Step											:= 1;
	eState											:= eWarmup;																// Set state
ELSIF rtrigEvacuation.Q THEN
	bEvacuationDone									:= FALSE;
	i2Step											:= 1;
	eState											:= eEvacuation;
ELSIF rtrigSteamBypass.Q THEN
	bSteamBypassDone								:= FALSE;
	i3Step											:= 1;
	eState											:= eSteamBypass;
ELSIF rtrigDesorption.Q THEN
	bDesorptionDone									:= FALSE;
	i4Step											:= 1;
	eState											:= eDesorption;
ELSIF rtrigRepressurization.Q THEN
	bRepressurizationDone							:= FALSE;
	i5Step											:= 1;
	eState											:= eRepressurization;
ELSIF rtrigAdsorption.Q THEN																								// Adsorption triggered
	bAdsorptionDone									:= FALSE;																// Clear Done flag
	bFanError										:= FALSE;
	i6Step											:= 1;																	// Start Adsorption Case statement
	eState											:= eAdsorption;															// Set state
END_IF

bDrainOn 											:= eState >= eWarmup AND eState <= eAdsorption;							// Turn on drain function

CASE eState OF
	
	eIdle:
		tgi_Machine_State							:= eIdle;																// Indicate state to HMI
		tgb_Auto_Mode								:= FALSE;																// Clear flags
		tgb_Stop_Cycle								:= FALSE;
		i1Step										:= 0;
		i2Step										:= 0;
		i3Step										:= 0;
		i4Step										:= 0;
		i5Step										:= 0;
		i6Step										:= 0;
		tgi_Current_Step							:= 0;
		IF bRunEvacuation THEN
			tgi_Machine_State						:= eEvacuation;
		ELSE
			tgi_Status								:= SEL(tgb_Test_Running, SEL(NOT tgb_Warmup_Complete, eSystem_Ready, eStart_Warm_Up), eTest_Running);
		END_IF
		
	eWarmup:
		tgi_Status									:= SEL(bStop, eWarmup_Running, eStopping_Warmup);
		IF tgb_Stop_Cycle THEN																							
			bStop									:= TRUE;
		ELSIF bWarmUpDone THEN																								// Process complete
			bStop									:= FALSE;
			IF tgb_Warmup_Complete THEN
				eState								:= eIdle;																// Return to manual state
			ELSE
				eState								:= ePause;																// User stopped - allow status string to be displayed momentarily
			END_IF	
		END_IF
		
	eEvacuation:
		tgi_Status									:= SEL(bStop, eEvacuation_Running, SEL(tgb_Auto_Mode, eStopping_Evacuation, eStopping_Process));
		IF tgb_Stop_Cycle THEN
			bStop									:= TRUE;			
		ELSIF bEvacuationDone THEN
			IF tgb_Auto_Mode THEN
				tgi_Machine_State					:= eSteamBypass;
			ELSE
				IF bStop THEN
					bStop							:= FALSE;
					eState							:= eIdle;
				ELSE
					tgi_Status						:= eEvacuation_Complete;
					bRunEvacuation					:= FALSE;
					eState							:= ePause;
				END_IF
			END_IF
		END_IF
		
	eSteamBypass:
		tgi_Status									:= SEL(bStop, eSteamBypass_Running, SEL(tgb_Auto_Mode, eStopping_SteamBypass, eStopping_Process));
		IF tgb_Stop_Cycle THEN
			bStop									:= TRUE;
		ELSIF bSteamBypassDone THEN
			IF tgb_Auto_Mode THEN
				tgi_Machine_State					:= eDesorption;
			ELSE
				IF bStop THEN
					bStop							:= FALSE;
					eState							:= eIdle;
				ELSE
					tgi_Status						:= eSteamBypass_Complete;
					eState							:= ePause;
				END_IF
			END_IF
		END_IF
		
	eDesorption:
		tgi_Status									:= SEL(bStop, eDesorption_Running, SEL(tgb_Auto_Mode, eStopping_Desorption, eStopping_Process));
		IF tgb_Stop_Cycle THEN
			bStop									:= TRUE;
		ELSIF bDesorptionDone THEN
			IF tgb_Auto_Mode THEN
				tgi_Machine_State					:= eRepressurization;
			ELSE
				IF bStop THEN
					bStop							:= FALSE;
					eState							:= eIdle;
				ELSE
					tgi_Status						:= eDesorption_Complete;
					eState							:= ePause;
				END_IF
			END_IF
		END_IF
		
	eRepressurization:
		tgi_Status									:= SEL(bStop, eRepressurization_Running, SEL(tgb_Auto_Mode, eStopping_Repressurization, eStopping_Process));
		IF tgb_Stop_Cycle THEN
			bStop									:= TRUE;
		ELSIF bRepressurizationDone THEN
			IF tgb_Auto_Mode THEN
				tgi_Machine_State					:= eAdsorption;
			ELSE
				IF bStop THEN
					bStop							:= FALSE;
					eState							:= eIdle;
				ELSE
					tgi_Status						:= eRepressurization_Complete;
					eState							:= ePause;
				END_IF
			END_IF
		END_IF
		
	eAdsorption:
		tgi_Status									:= SEL(bStop, eAdsorption_Running, SEL(tgb_Auto_Mode, eStopping_Adsorption, eStopping_Process));
		IF tgb_Stop_Cycle THEN
			bStop									:= TRUE;
		ELSIF bAdsorptionDone THEN
			IF tgb_Auto_Mode THEN
				tgi_Cycle_Count						:= tgi_Cycle_Count + 1;
				gpdiCycle_Count						:= gpdiCycle_Count + 1;
				IF tgi_Cycle_Count >= tgi_Cycles_To_Run THEN
					eState							:= eIdle;
				ELSE
					tgi_Machine_State				:= eEvacuation;
				END_IF
			ELSE
				IF bFanError THEN
					tgi_Machine_State				:= eEvacuation;
				ELSIF bStop THEN
					bStop							:= FALSE;
					eState							:= eIdle;
				ELSIF bRunEvacuation THEN
					eState							:= eIdle;
				ELSE
					tgi_Status						:= eAdsorption_Complete;
					eState							:= ePause;
				END_IF
			END_IF
		END_IF
		
	eReset:
		IF tonReset.Q THEN
			A0_Reset();
			eState									:= eIdle;
		END_IF

	ePause:
		tgi_Machine_State							:= ePause;
		IF tonPause.Q THEN
			eState									:= eIdle;
		END_IF
		
	eSystemError:
		;
		
END_CASE

CASE tgi_Alarm_State OF
	
	1: ;																					// Level 1 alarm 
	
	2: ;																					// Level 2 alarm
	
	3: 	tgb_Stop_Cycle								:= TRUE;								// Level 3 alarm - stop cycle but no reset
		tgi_Alarm_State								:= 5;
	
	4:	tgb_Warmup_Complete							:= FALSE;								// Level 4 alarm - reset everything
		A0_Reset();
		tgi_Alarm_State								:= 5;
		eState										:= eSystemError;

	5:	 ;
	
END_CASE

rtrigStatusReady(CLK:= tgb_Warmup_Complete);
IF rtrigStatusReady.Q THEN
	tgi_Status										:= eSystem_Ready;
END_IF

A1_WarmUp();																										// Run action for this state
A2_Evacuation();
A3_SteamBypass();
A4_Desorption();
A5_Repressurization();
A6_Adsorption();

tonTimer1(IN:= bTimer1, PT:= REAL_TO_TIME(rTime1));
tonTimer2(IN:= bTimer2, PT:= REAL_TO_TIME(rTime2));

IF i1Step + i2Step + i3Step + i4Step + i5Step + i6Step > 0 THEN
	IF bTimer1 THEN
		tgr_Remaining_Time							:= rTime1 - TIME_TO_REAL(tonTimer1.ET);
	ELSIF bTimer2 THEN
		tgr_Remaining_Time							:= rTime2 - TIME_TO_REAL(tonTimer2.ET);
	ELSE
		tgr_Remaining_Time							:= 0;
	END_IF
END_IF

tgs_Status											:= strStatusLabel[tgi_Status];
bRunning											:= eState > eIdle AND eState < eReset;									// 09/19/23 PS
gbVFDTest											:= SEL(bRunning, gbVFDTest, FALSE);										// 09/19/23 PS
tgb_Drains_On										:= SEL(tgb_Auto_Mode, tgb_Drains_On, FALSE);							// 09/19/23 PS

tonReset(IN:= eState = eReset, PT:= REAL_TO_TIME(RESET_TIME));
tonPause(IN:= eState = ePause, PT:= REAL_TO_TIME(RESET_TIME));

ACTION A_ClearProcess:
// Calvin - A_ClearProcess
// Rev 1.00 - September 22, 2023

IF giActiveAlarm > 0 THEN
	gsAlarmInfo[giActiveAlarm]				:= CONCAT(INT_TO_STRING(iStep), strError);
	gbAlarmsLoaded							:= FALSE;
END_IF
bTimer1								 		:= FALSE;
bTimer2								 		:= FALSE;
tgb_Stop_Cycle								:= FALSE;
tgb_Auto_Mode								:= FALSE;
END_ACTION

ACTION A_DPT_Fan_Test:
// Calvin - A_DPT_Fan_Test
// Rev 1.00 - July 14, 2023

rtrigFanTest(CLK:= tgb_Test_Mode);
ftrigFanTest(CLK:= tgb_Test_Mode);

IF rtrigFanTest.Q THEN
	iFanTestStep									:= 1;
END_IF
IF ftrigFanTest.Q THEN
	iFanTestStep									:= 4;
END_IF

CASE iFanTestStep OF
	
	0:	tgb_Test_Running							:= FALSE;

	1:	tgr_IP_1102A								:= 100;
		tgr_IP_1102B								:= 100;
		tgb_Test_Running							:= TRUE;
		rFanIncrement								:= 10;
		tgr_HS_1102									:= 0;
		iFanTestStep								:= 2;
	
	2:	IF tgb_IP_1102A_Open AND tgb_IP_1102B_Open THEN
			bFanTimer								:= TRUE;
			tgr_HS_1102								:= rFanIncrement;
			iFanTestStep							:= 3;
		END_IF
		
	3:	;
	
	4:	bFanTimer									:= FALSE;
		tgr_HS_1102									:= 0;
		IF tgr_HS_1102_RPM = 0 THEN
			tgr_IP_1102A							:= 0;
			tgr_IP_1102B							:= 0;
			iFanTestStep							:= 0;
		END_IF

END_CASE;

IF tonFanTest.Q THEN
	tgr_HS_1102										:= tgr_HS_1102 + rFanIncrement;
	IF tgr_HS_1102 > rFanMaximum THEN
		rFanIncrement								:= 0 - rFanIncrement;
		tgr_HS_1102									:= rFanMaximum + rFanIncrement;
	ELSIF tgr_HS_1102 <= 0 THEN
		tgb_Test_Mode								:= FALSE;
	END_IF
	
	tonFanTest(IN:= FALSE);
END_IF

tonFanTest(IN:= bFanTimer, PT:= tFanTestTime);
END_ACTION

ACTION A_Inputs_Outputs:
// Calvin - A_Inputs_Outputs
// Rev 1.00 - September 20, 2023

//// DIGITAL IN
tgb_HS_1104_Open									:= ZSH_1104;			
tgb_HS_1104_Closed									:= ZSL_1104;				
tgb_HS_1107_Open									:= ZSH_1107;			
tgb_HS_1107_Closed									:= ZSL_1107;				
tgb_HS_1101A_Open									:= ZSH_1101A;				
tgb_HS_1101A_Closed									:= ZSL_1101A;				
tgb_HS_1101B_Open									:= ZSH_1101B;				
tgb_HS_1101B_Closed									:= ZSL_1101B;			
tgb_HS_1201_LSH										:= LSH_1201;					
tgb_HS_1201_LSL										:= LSL_1201;					
tgb_HS_1103A_Open									:= ZSH_1103A;				
tgb_HS_1103A_Closed									:= ZSL_1103A;				
tgb_HS_1103B_Open									:= ZSH_1103B;				
tgb_HS_1103B_Closed									:= ZSL_1103B;				
tgb_HS_1202_LSH										:= LSH_1202;			
tgb_HS_1202_LSL										:= LSL_1202;				
tgb_HS_1302A_Open									:= ZSH_1302A;			
tgb_HS_1302A_Closed									:= ZSL_1302A;			
tgb_HS_1301A_Open									:= ZSH_1301A;				
tgb_HS_1301A_Closed									:= ZSL_1301A;				
tgb_HS_1301B_Open									:= ZSH_1301B;				
tgb_HS_1301B_Closed									:= ZSL_1301B;				
tgb_HS_1300B_Open									:= ZSH_1300;					
tgb_HS_1300B_Closed									:= ZSL_1300;					
tgb_HS_1300A_LSH									:= LSH_1300A;			
tgb_HS_1300A_LSL									:= LSL_1300A;				
tgb_SV_1201_Open									:= ZSH_1202;				
tgb_SV_1201_Closed									:= ZSL_1202;				

//// ANALOG IN
tgr_DPT_1102A										:= F_AnalogIn(DPT_1102A, DPT_1102A_LOW, DPT_1102A_HIGH, DPT_1102A_MIN, DPT_1102A_OFFSET);
tgr_FIC_1102										:= F_AnalogIn(FIC_1102, FIC_1102_LOW, FIC_1102_HIGH, FIC_1102_MIN, FIC_1102_OFFSET);
tgr_AI_1102A										:= F_AnalogIn(AI_1102A, AI_1102A_LOW, AI_1102A_HIGH, AI_1102A_MIN, AI_1102A_OFFSET);
tgr_MI_1102A										:= F_AnalogIn(MI_1102A, MI_1102A_LOW, MI_1102A_HIGH, MI_1102A_MIN, MI_1102A_OFFSET);
tgr_ZT_1102A										:= F_AnalogIn(ZT_1102A, ZT_1102A_LOW, ZT_1102A_HIGH, ZT_1102A_MIN, ZT_1102A_OFFSET);
tgr_PI_1100											:= F_AnalogIn(PI_1100, PI_1100_LOW, PI_1100_HIGH, PI_1100_MIN, PI_1100_OFFSET);
tgr_DPT_1100										:= F_AnalogIn(DPT_1100, DPT_1100_LOW, DPT_1100_HIGH, DPT_1100_MIN, DPT_1100_OFFSET);
tgr_ZT_1102B										:= F_AnalogIn(ZT_1102B, ZT_1102B_LOW, ZT_1102B_HIGH, ZT_1102B_MIN, ZT_1102B_OFFSET);
tgr_AI_1102B										:= F_AnalogIn(AI_1102B, AI_1102B_LOW, AI_1102B_HIGH, AI_1102B_MIN, AI_1102B_OFFSET);
tgr_MI_1102B										:= F_AnalogIn(MI_1102B, MI_1102B_LOW, MI_1102B_HIGH, MI_1102B_MIN, MI_1102B_OFFSET);
tgr_DPT_1102B										:= F_AnalogIn(DPT_1102B, DPT_1102B_LOW, DPT_1102B_HIGH, DPT_1102B_MIN, DPT_1102B_OFFSET);
tgr_FI_1200_1										:= F_AnalogIn(FI_1200_1, FI_1200_1_LOW, FI_1200_1_HIGH, FI_1200_1_MIN, FI_1200_1_OFFSET);
tgr_FI_1200_2										:= F_AnalogIn(FI_1200_2, FI_1200_2_LOW, FI_1200_2_HIGH, FI_1200_2_MIN, FI_1200_2_OFFSET);
tgr_FI_1200_3										:= F_AnalogIn(FI_1200_3, FI_1200_3_LOW, FI_1200_3_HIGH, FI_1200_3_MIN, FI_1200_3_OFFSET);
tgr_FI_1201_1										:= F_AnalogIn(FI_1201_1, FI_1201_1_LOW, FI_1201_1_HIGH, FI_1201_1_MIN, FI_1201_1_OFFSET);
tgr_FI_1201_2										:= F_AnalogIn(FI_1201_2, FI_1201_2_LOW, FI_1201_2_HIGH, FI_1201_2_MIN, FI_1201_2_OFFSET);
tgr_FI_1201_3										:= F_AnalogIn(FI_1201_3, FI_1201_3_LOW, FI_1201_3_HIGH, FI_1201_3_MIN, FI_1201_3_OFFSET);
tgr_PI_1200											:= F_AnalogIn(PI_1200, PI_1200_LOW, PI_1200_HIGH, PI_1200_MIN, PI_1200_OFFSET);
tgr_PI_1001											:= F_AnalogIn(PI_1001, PI_1001_LOW, PI_1001_HIGH, PI_1001_MIN, PI_1001_OFFSET);
tgr_FI_1001											:= F_AnalogIn(FI_1001, FI_1001_LOW, FI_1001_HIGH, FI_1001_MIN, FI_1001_OFFSET);
tgr_ZT_1101											:= F_AnalogIn(ZT_1101, ZT_1101_LOW, ZT_1101_HIGH, ZT_1101_MIN, ZT_1101_OFFSET);
tgr_PI_1101											:= F_AnalogIn(PI_1101, PI_1101_LOW, PI_1101_HIGH, PI_1101_MIN, PI_1101_OFFSET);
tgr_LI_1204											:= F_AnalogIn(LI_1204, LI_1204_LOW, LI_1204_HIGH, LI_1204_MIN, LI_1204_OFFSET);
tgr_PI_1300											:= F_AnalogIn(PI_1300, PI_1300_LOW, PI_1300_HIGH, PI_1300_MIN, PI_1300_OFFSET);
tgr_LIC_1300										:= F_AnalogIn(LIC_1300, LIC_1300_LOW, LIC_1300_HIGH, LIC_1300_MIN, LIC_1300_OFFSET);
tgr_FI_1300											:= F_AnalogIn(FI_1300, FI_1300_LOW, FI_1300_HIGH, FI_1300_MIN, FI_1300_OFFSET);
tgr_FI_1301											:= F_AnalogIn(FI_1301, FI_1301_LOW, FI_1301_HIGH, FI_1301_MIN, FI_1301_OFFSET);
tgr_AI_1301											:= F_AnalogIn(AI_1301, AI_1301_LOW, AI_1301_HIGH, AI_1301_MIN, AI_1301_OFFSET);
tgr_ZT_1302B										:= F_AnalogIn(ZT_1302B, ZT_1302B_LOW, ZT_1302B_HIGH, ZT_1302B_MIN, ZT_1302B_OFFSET);
tgr_MI_2001											:= F_AnalogIn(MI_2001, MI_2001_LOW, MI_2001_HIGH, MI_2001_MIN, MI_2001_OFFSET);
tgr_TI_2001											:= F_AnalogIn(TI_2001, TI_2001_LOW, TI_2001_HIGH, TI_2001_MIN, TI_2001_OFFSET);
tgr_SI_2001											:= F_AnalogIn(SI_2001, SI_2001_LOW, SI_2001_HIGH, SI_2001_MIN, SI_2001_OFFSET);
tgr_ZI_2001											:= F_AnalogIn(ZI_2001, ZI_2001_LOW, ZI_2001_HIGH, ZI_2001_MIN, ZI_2001_OFFSET);
tgr_PI_2001											:= F_AnalogIn(PI_2001, PI_2001_LOW, PI_2001_HIGH, PI_2001_MIN, PI_2001_OFFSET);
tgr_ZXI_2002										:= F_AnalogIn(WORD_TO_INT(ZXI_2002), ZXI_2002_LOW, ZXI_2002_HIGH, ZXI_2002_MIN, ZXI_2002_OFFSET);		
tgr_ZYI_2002										:= F_AnalogIn(WORD_TO_INT(ZYI_2002), ZYI_2002_LOW, ZYI_2002_HIGH, ZYI_2002_MIN, ZYI_2002_OFFSET);		
tgr_IT_1											:= F_Current(IT_1);
tgr_IT_2											:= F_Current(IT_2); 
tgr_IT_3											:= F_Current(IT_3); 
tgr_VT_1											:= F_Voltage(VT_1);
tgr_VT_2											:= F_Voltage(VT_2);
tgr_VT_3											:= F_Voltage(VT_3);

//// DIGITAL OUT
YL_1001												:= tgb_YL_1001;
tgb_YL_1001_On										:= YL_1001; 
YL_1002												:= YL_1001;										// YL_1002 is triggered whenever YL_1001 is triggered
HS_1107												:= tgb_HS_1107;	
tgb_HS_1107_On										:= HS_1107;			
HS_1101A											:= tgb_HS_1101A;
tgb_HS_1101A_On										:= HS_1101A;
HS_1101B											:= tgb_HS_1101B;
tgb_HS_1101B_On										:= HS_1101B;				
HS_1201												:= tgb_HS_1201;
tgb_HS_1201_On										:= HS_1201;				
AI_1102A_Pump										:= tgb_AI_1102A_Pump OR bRunning;										// 09/19/23 PS
tgb_AI_1102A_Pump_On								:= AI_1102A_Pump;
AI_1102A_Solenoid									:= NOT tgb_AI_1102A_Solenoid AND NOT bRunning;							// 09/19/23 PS
tgb_AI_1102A_Solenoid_On							:= NOT AI_1102A_Solenoid;													
AI_1102B_Pump										:= tgb_AI_1102B_Pump OR bRunning;										// 09/19/23 PS
tgb_AI_1102B_Pump_On								:= AI_1102B_Pump;
AI_1102B_Solenoid									:= NOT tgb_AI_1102B_Solenoid AND NOT bRunning;							// 09/19/23 PS			
tgb_AI_1102B_Solenoid_On							:= NOT AI_1102B_Solenoid;													
HS_1103A											:= tgb_HS_1103A;
tgb_HS_1103A_On										:= HS_1103A;				
HS_1103B											:= tgb_HS_1103B;
tgb_HS_1103B_On										:= HS_1103B;				
HS_1202												:= tgb_HS_1202;	
tgb_HS_1202_On										:= HS_1202;			
HS_1203												:= tgb_HS_1203;				
tgb_HS_1203_On										:= HS_1203;				
HS_1200												:= tgb_HS_1200;				
tgb_HS_1200_On										:= HS_1200;
SV_1201												:= tgb_SV_1201;												// 09/19/23 PS	
tgb_SV_1201_On										:= SV_1201;			
HS_1302A											:= tgb_HS_1302A;
tgb_HS_1302A_On										:= HS_1302A;				
HS_1301A											:= tgb_HS_1301A;
tgb_HS_1301A_On										:= HS_1301A;				
HS_1301												:= tgb_HS_1301;
tgb_HS_1301_On										:= HS_1301;				
HS_1301B											:= tgb_HS_1301B;
tgb_HS_1301B_On										:= HS_1301B;			
HS_1300A											:= tgb_HS_1300A;
tgb_HS_1300A_On										:= HS_1300A;			
HS_1300B											:= tgb_HS_1300B;
tgb_HS_1300B_On										:= HS_1300B;				
HS_1305												:= tgb_HS_1305;
tgb_HS_1305_On										:= HS_1305;
HS_1104												:= tgb_HS_1104;
tgb_HS_1104_On										:= HS_1104;

//// ANALOG OUT
IF bRunValveModulation THEN
	IF tgr_PI_1100 >= tgr_SP_IP_1302B_Reactor_High THEN
		tgr_IP_1302B								:= tgr_SP_IP_1302B_Valve_Low;
	ELSIF tgr_PI_1100 <= tgr_SP_IP_1302B_Reactor_Low THEN
		tgr_IP_1302B								:= tgr_SP_IP_1302B_Valve_High;
	END_IF
	bValveInRange									:= tgr_PI_1100 >= tgr_SP_IP_1302B_Reactor_Low AND tgr_PI_1100 <= tgr_SP_IP_1302B_Reactor_High;
END_IF
		
tgb_IP_1102A_Open									:= tgr_ZT_1102A > (BV_OPEN_MAX - BV_OPEN_POS_THRESHOLD);
tgb_IP_1102A_Closed									:= tgr_ZT_1102A < BV_CLOSED_POS_THRESHOLD;
tgb_IP_1102B_Open									:= tgr_ZT_1102B > (BV_OPEN_MAX - BV_OPEN_POS_THRESHOLD);
tgb_IP_1102B_Closed									:= tgr_ZT_1102B < BV_CLOSED_POS_THRESHOLD;
gbHS_1102ValvesOpen									:= tgb_IP_1102A_Open AND tgb_IP_1102B_Open;
gbHS_1102ValvesClosed								:= tgb_IP_1102A_Closed AND tgb_IP_1102B_Closed;

gbRunVFD											:= TRUE;
HS_1102_Enable										:= gbRunVFD;		
grHS_1102Out										:= SEL(NOT tgb_HS_1102_Enabled OR NOT gbHS_1102ValvesOpen, tgr_HS_1102, 0);
HS_1102_Out											:= REAL_TO_INT(grHS_1102Out * PERCENT_FACTOR);
tgr_HS_1102_Output									:= grHS_1102Out;

IP_1302B											:= REAL_TO_INT(tgr_IP_1302B * PERCENT_FACTOR);
tgr_IP_1302B_Output									:= tgr_IP_1302B;
IP_1101												:= REAL_TO_INT(tgr_IP_1101 * PERCENT_FACTOR);
tgr_IP_1101_Output									:= tgr_IP_1101;
IP_1102A											:= REAL_TO_INT(tgr_IP_1102A * PERCENT_FACTOR);
tgr_IP_1102A_Output									:= tgr_IP_1102A;
IP_1102B											:= REAL_TO_INT(tgr_IP_1102B * PERCENT_FACTOR);
tgr_IP_1102B_Output									:= tgr_IP_1102B;
         
LED1_G												:= SEL(tgb_IP_1102A_Open, SEL(tgb_IP_1102A_Closed, tgb_Half_Sec_Pulse, FALSE), TRUE); 
LED1_R												:= NOT LED1_G;
LED1_Buzzer											:= NOT tgb_IP_1102A_Open AND NOT tgb_IP_1102A_Closed; 
LED2_G												:= SEL(tgb_IP_1102B_Open, SEL(tgb_IP_1102B_Closed, tgb_Half_Sec_Pulse, FALSE), TRUE); 
LED2_R												:= NOT LED2_G; 
LED2_Buzzer											:= NOT tgb_IP_1102B_Open AND NOT tgb_IP_1102B_Closed; 


// Lightbar
IF tgb_Active_Alarm OR NOT tgb_ADS_Active THEN
	LED3_R											:= tgb_Half_Sec_Pulse;
	LED3_Y											:= FALSE;
	LED3_G											:= FALSE;
ELSIF eState = eReset OR eState = eIdle THEN
	LED3_R											:= FALSE;
	LED3_Y											:= TRUE;
	LED3_G											:= FALSE;
ELSE
	LED3_R											:= FALSE;
	LED3_Y											:= FALSE;
	LED3_G											:= TRUE;
END_IF

tgi_Total_Cycle_Count								:= gpdiCycle_Count;
END_ACTION

ACTION A_Interlocks:
// Calvin - A_Interlocks
// Rev 1.00 - September 19, 2023
END_ACTION

ACTION A_Modbus_Points:
// Calvin - A_Modbus_Points
// Rev 1.00 - April 7, 2023

IF iMBPFunction = 0 THEN															// Modbus is not busy
	IF gbReadMBWeather THEN
		MBP_Master.UnitID 							:= 1;							// Weather Station Modbus address
		wMBPAddress									:= 8193;
		wMBPQuantity								:= 1;
		bMBPWeather									:= TRUE;
		iMBPFunction								:= eMBReadRegs;
	ELSIF gbReadMBInclinometer THEN
		MBP_Master.UnitID 							:= 80;							// Inclinometer Modbus address
		wMBPAddress									:= 61;
		wMBPQuantity								:= 2;
		bMBPWeather									:= FALSE;
		iMBPFunction								:= eMBReadRegs;
	END_IF
	IF bMBPWeather THEN
		; 	// Get weather values here
	ELSE
		ZXI_2002									:= wMBPReadData[0];
		ZYI_2002									:= wMBPReadData[1];
	END_IF
ELSIF tonMBPReset.Q THEN
	iMBPFunction									:= eMBIdle;
END_IF
tonMBPReset(IN:= iMBPFunction > 0, PT:= MODBUS_TIMEOUT);

CASE iMBPFunction OF
	
	eMBIdle:
		MBP_Master.Execute 							:= FALSE;
		
	eMBReadRegs:
		MBP_Master.ReadRegs(
			Quantity								:= wMBPQuantity, 
			MBAddr									:= wMBPAddress, 
			cbLength								:= SIZEOF(wMBPReadData), 
			pMemoryAddr								:= ADR(wMBPReadData), 
			Execute									:= TRUE, 
			Timeout									:= MODBUS_TIMEOUT, 
			BUSY									=> bMBPBusy, 
			Error									=> bMBPError, 
			ErrorId									=> MBP_Errors, 
			cbRead									=> uiMBPRead);
		MBP_Master.ReadRegs(BUSY=> bMBPBusy);
		IF NOT MBP_Master.BUSY THEN
			MBP_Master.Execute 						:= FALSE;
			MBP_Master.ReadRegs(BUSY=> bMBPBusy);
			IF MBP_Master.Error THEN
				MBP_Master.ReadRegs();
			ELSE
				iMBPFunction 						:= 0;			
			END_IF
		END_IF
	
	ELSE
		iMBPFunction 								:= 0;
	
END_CASE
END_ACTION

ACTION A_Modbus_VFD:
// Calvin - A_Modbus_VFD
// Rev 1.00 - July 3, 2023

MBV_Master.UnitID 									:= 1;														// VFD address is 1

IF iMBVFunction = 0 THEN																						// Modbus is not busy
	IF gbReadMBVFD THEN
		gbReadMBVFD									:= FALSE;
		wMBVAddress									:= MB_VFD_BLOCK_ADDR;										// Read Block parameters
		wMBVQuantity								:= 4;														// Read status, current frequency, current rpm
		iMBVFunction								:= eMBReadRegs;
		bMBVStatusCheck								:= FALSE;
	END_IF
	tgb_HS_1102_Enabled								:= (wMBVReadData[0] AND wMBVStatus) <> 0;
	tgr_HS_1102_RPM									:= WORD_TO_REAL(wMBVReadData[2]);
	tgr_HS_1102_RPM									:= SEL(tgr_HS_1102_RPM < 20, tgr_HS_1102_RPM, 0);
	tgr_HS_1102V									:= WORD_TO_REAL(wMBVReadData[1]);
	tgb_HS_1102_Running								:= tgb_HS_1102_Enabled AND tgr_HS_1102_RPM > 20;
ELSIF tonMBVReset.Q THEN																						// Reset Modbus routine if still active after timeout
	iMBVFunction									:= 0;	
END_IF
tonMBVReset(IN:= iMBVFunction > 0, PT:= MODBUS_TIMEOUT);

CASE iMBVFunction OF
	
	eMBIdle:
		MBV_Master.Execute 							:= FALSE;
		
	eMBReadRegs:
		MBV_Master.ReadRegs(
			Quantity								:= wMBVQuantity, 
			MBAddr									:= wMBVAddress, 
			cbLength								:= SIZEOF(wMBVReadData), 
			pMemoryAddr								:= ADR(wMBVReadData), 
			Execute									:= TRUE, 
			Timeout									:= MODBUS_TIMEOUT, 
			BUSY									=> bMBVBusy, 
			Error									=> bMBVError, 
			ErrorId									=> MBV_Errors, 
			cbRead									=> uiMBVRead);
		MBV_Master.ReadRegs(BUSY=> bMBVBusy);
		IF NOT MBV_Master.BUSY THEN
			MBV_Master.Execute 						:= FALSE;
			MBV_Master.ReadRegs(BUSY=> bMBVBusy);
			IF MBV_Master.Error THEN
				MBV_Master.ReadRegs();
			ELSE
				iMBVFunction 						:= 0;			
			END_IF
		END_IF
	
	eMBWriteSingleReg:	
		MBV_Master.WriteSingleRegister(
			Quantity								:= wMBVQuantity, 
			MBAddr									:= wMBVAddress, 
			cbLength								:= SIZEOF(wMBVWriteData), 
			pMemoryAddr								:= ADR(wMBVWriteData), 
			Execute									:= TRUE, 
			Timeout									:= MODBUS_TIMEOUT, 
			BUSY									=> bMBVBusy, 
			Error									=> bMBVError, 
			ErrorId									=> MBV_Errors, 
			cbRead									=> uiMBVRead);
		MBV_Master.WriteSingleRegister(BUSY=> bMBVBusy);
		IF NOT MBV_Master.BUSY THEN
			MBV_Master.Execute 						:= FALSE;
			MBV_Master.WriteSingleRegister(BUSY=> bMBVBusy);
			IF MBV_Master.Error THEN
				MBV_Master.WriteSingleRegister();
			ELSE
				iMBVFunction 						:= 0;			
			END_IF
		END_IF


// These are not currently used	

	eMBReadCoils:
		MBV_Master.ReadCoils(
			Quantity								:= wMBVQuantity, 
			MBAddr									:= wMBVAddress, 
			cbLength								:= SIZEOF(wMBVReadData), 
			pMemoryAddr								:= ADR(wMBVReadData), 
			Execute									:= TRUE, 
			Timeout									:= MODBUS_TIMEOUT, 
			BUSY									=> bMBVBusy, 
			Error									=> bMBVError, 
			ErrorId									=> MBV_Errors, 
			cbRead									=> uiMBVRead);
		MBV_Master.ReadCoils(BUSY=> bMBVBusy);
		IF NOT MBV_Master.BUSY THEN
			MBV_Master.Execute 						:= FALSE;
			MBV_Master.ReadCoils(BUSY=> bMBVBusy);
			IF MBV_Master.Error THEN
				MBV_Master.ReadCoils();
			ELSE
				iMBVFunction 						:= 0;			
			END_IF
		END_IF
	
